ABB RAPID module: P802.mod

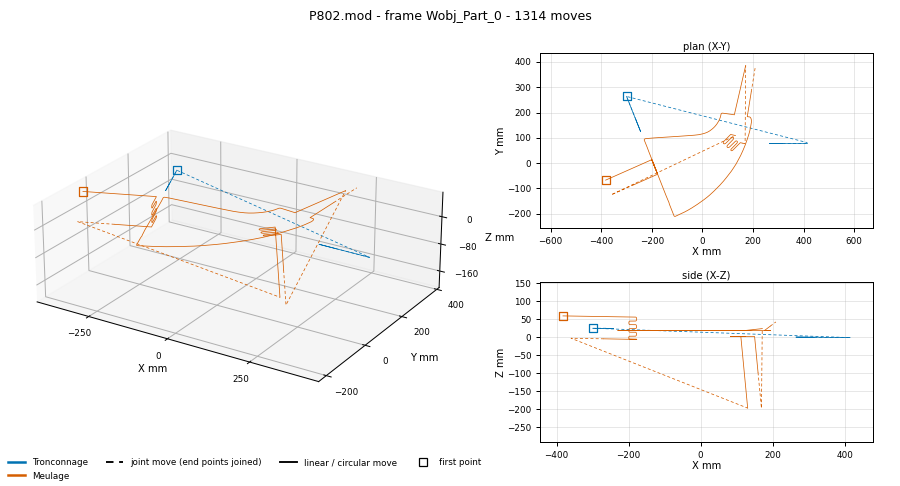
[picture p0: tool path of P802.mod in frame Wobj_Part_0, 1314 of 1328 moves have a stored position in this frame; points joined in program order, loops and branches not executed]
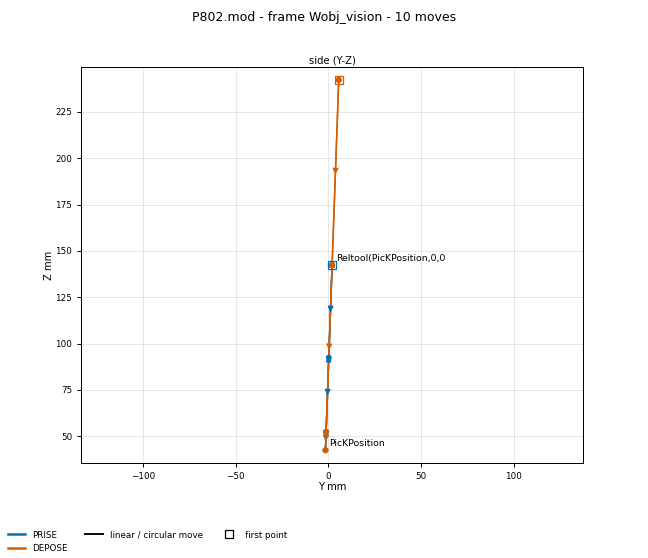
[picture p1: tool path of P802.mod in frame Wobj_vision, 10 of 1328 moves have a stored position in this frame; points joined in program order, loops and branches not executed]
MODULE P802

    ! Nom         :P802
    ! Description :
    ! Créé le     :31/05/2023 09:39:48

    LOCAL CONST SPEEDDATA VitesseLente :=[3,500,0,0];
	LOCAL CONST SPEEDDATA VitesseRapide :=[30,500,0,0];
	LOCAL CONST SPEEDDATA VitesseTronconnage :=[2,500,0,0];
	LOCAL CONST SPEEDDATA VitesseTronconnageApp :=[10,500,0,0];
    !
    !Point de prise
    LOCAL PERS Robtarget PicKPosition := [[-42.0484766120473,-1.61957801853713,42.4060496277998],[0.0147319075907155,0.941094234914177,-0.337609036243247,0.0120312325612993],[0,0,0,0],[8.999999E+09,8.999999E+09,8.999999E+09,8.999999E+09,8.999999E+09,8.999999E+09]];
	LOCAL PERS Pose Ref := [[0,0,0],[1,0,0,0]];
    !
    !Declaration des points de meulage

    !Tr_meulage_motif_1 : Meulage d'un motif
    LOCAL CONST Robtarget Tr_meulage_motif_1_0 := [[-199.5515,14.0755400390625,55.70646484375],[0.587839766788017,-0.597604018313253,0.388723125784971,-0.382371778977509],[0,0,0,0],[8.999999E+09,8.999999E+09,8.999999E+09,8.999999E+09,8.999999E+09,8.999999E+09]];
    LOCAL CONST Robtarget Tr_meulage_motif_1_1 := [[-199.1803125,13.146982421875,55.70646484375],[0.587839766788017,-0.597604018313253,0.388723125784971,-0.382371778977509],[0,0,0,0],[8.999999E+09,8.999999E+09,8.999999E+09,8.999999E+09,8.999999E+09,8.999999E+09]];
    LOCAL CONST Robtarget Tr_meulage_motif_1_2 := [[-198.809125,12.2184248046875,55.70646484375],[0.587839766788017,-0.597604018313253,0.388723125784971,-0.382371778977509],[0,0,0,0],[8.999999E+09,8.999999E+09,8.999999E+09,8.999999E+09,8.999999E+09,8.999999E+09]];
    LOCAL CONST Robtarget Tr_meulage_motif_1_3 := [[-198.4379375,11.2898671875,55.70646875],[0.587839766788017,-0.597604018313253,0.388723125784971,-0.382371778977509],[0,0,0,0],[8.999999E+09,8.999999E+09,8.999999E+09,8.999999E+09,8.999999E+09,8.999999E+09]];
    LOCAL CONST Robtarget Tr_meulage_motif_1_4 := [[-198.06675,10.36130859375,55.70646875],[0.587839766788017,-0.597604018313253,0.388723125784971,-0.382371778977509],[0,0,0,0],[8.999999E+09,8.999999E+09,8.999999E+09,8.999999E+09,8.999999E+09,8.999999E+09]];
    LOCAL CONST Robtarget Tr_meulage_motif_1_5 := [[-197.6955625,9.4327509765625,55.70646875],[0.587839766788017,-0.597604018313253,0.388723125784971,-0.382371778977509],[0,0,0,0],[8.999999E+09,8.999999E+09,8.999999E+09,8.999999E+09,8.999999E+09,8.999999E+09]];
    LOCAL CONST Robtarget Tr_meulage_motif_1_6 := [[-197.324375,8.504193359375,55.70646875],[0.587839766788017,-0.597604018313253,0.388723125784971,-0.382371778977509],[0,0,0,0],[8.999999E+09,8.999999E+09,8.999999E+09,8.999999E+09,8.999999E+09,8.999999E+09]];
    LOCAL CONST Robtarget Tr_meulage_motif_1_7 := [[-196.9531875,7.57563525390625,55.70646875],[0.587839766788017,-0.597604018313253,0.388723125784971,-0.382371778977509],[0,0,0,0],[8.999999E+09,8.999999E+09,8.999999E+09,8.999999E+09,8.999999E+09,8.999999E+09]];
    LOCAL CONST Robtarget Tr_meulage_motif_1_8 := [[-196.582,6.64707763671875,55.70647265625],[0.587839766788017,-0.597604018313253,0.388723125784971,-0.382371778977509],[0,0,0,0],[8.999999E+09,8.999999E+09,8.999999E+09,8.999999E+09,8.999999E+09,8.999999E+09]];
    LOCAL CONST Robtarget Tr_meulage_motif_1_9 := [[-196.2108125,5.71852001953125,55.70647265625],[0.587839766788017,-0.597604018313253,0.388723125784971,-0.382371778977509],[0,0,0,0],[8.999999E+09,8.999999E+09,8.999999E+09,8.999999E+09,8.999999E+09,8.999999E+09]];
    LOCAL CONST Robtarget Tr_meulage_motif_1_10 := [[-195.839625,4.7899619140625,55.70647265625],[0.587839766788017,-0.597604018313253,0.388723125784971,-0.382371778977509],[0,0,0,0],[8.999999E+09,8.999999E+09,8.999999E+09,8.999999E+09,8.999999E+09,8.999999E+09]];
    LOCAL CONST Robtarget Tr_meulage_motif_1_11 := [[-195.4684375,3.861404296875,55.70647265625],[0.587839766788017,-0.597604018313253,0.388723125784971,-0.382371778977509],[0,0,0,0],[8.999999E+09,8.999999E+09,8.999999E+09,8.999999E+09,8.999999E+09,8.999999E+09]];
    LOCAL CONST Robtarget Tr_meulage_motif_1_12 := [[-195.09725,2.93284643554688,55.70647265625],[0.587839766788017,-0.597604018313253,0.388723125784971,-0.382371778977509],[0,0,0,0],[8.999999E+09,8.999999E+09,8.999999E+09,8.999999E+09,8.999999E+09,8.999999E+09]];
    LOCAL CONST Robtarget Tr_meulage_motif_1_13 := [[-194.7260625,2.00428857421875,55.7064765625],[0.587839766788017,-0.597604018313253,0.388723125784971,-0.382371778977509],[0,0,0,0],[8.999999E+09,8.999999E+09,8.999999E+09,8.999999E+09,8.999999E+09,8.999999E+09]];
    LOCAL CONST Robtarget Tr_meulage_motif_1_14 := [[-194.354875,1.07573071289063,55.7064765625],[0.587839766788017,-0.597604018313253,0.388723125784971,-0.382371778977509],[0,0,0,0],[8.999999E+09,8.999999E+09,8.999999E+09,8.999999E+09,8.999999E+09,8.999999E+09]];
    LOCAL CONST Robtarget Tr_meulage_motif_1_15 := [[-193.9836875,0.147172897338867,55.7064765625],[0.587839766788017,-0.597604018313253,0.388723125784971,-0.382371778977509],[0,0,0,0],[8.999999E+09,8.999999E+09,8.999999E+09,8.999999E+09,8.999999E+09,8.999999E+09]];
    LOCAL CONST Robtarget Tr_meulage_motif_1_16 := [[-193.6125,-0.781384948730469,55.7064765625],[0.587839766788017,-0.597604018313253,0.388723125784971,-0.382371778977509],[0,0,0,0],[8.999999E+09,8.999999E+09,8.999999E+09,8.999999E+09,8.999999E+09,8.999999E+09]];
    LOCAL CONST Robtarget Tr_meulage_motif_1_17 := [[-193.2413125,-1.70994274902344,55.70648046875],[0.587839766788017,-0.597604018313253,0.388723125784971,-0.382371778977509],[0,0,0,0],[8.999999E+09,8.999999E+09,8.999999E+09,8.999999E+09,8.999999E+09,8.999999E+09]];
    LOCAL CONST Robtarget Tr_meulage_motif_1_18 := [[-192.870125,-2.63850048828125,55.70648046875],[0.587839766788017,-0.597604018313253,0.388723125784971,-0.382371778977509],[0,0,0,0],[8.999999E+09,8.999999E+09,8.999999E+09,8.999999E+09,8.999999E+09,8.999999E+09]];
    LOCAL CONST Robtarget Tr_meulage_motif_1_19 := [[-192.4989375,-3.56705834960938,55.70648046875],[0.587839766788017,-0.597604018313253,0.388723125784971,-0.382371778977509],[0,0,0,0],[8.999999E+09,8.999999E+09,8.999999E+09,8.999999E+09,8.999999E+09,8.999999E+09]];
    LOCAL CONST Robtarget Tr_meulage_motif_1_20 := [[-192.12775,-4.4956162109375,55.70648046875],[0.587839766788017,-0.597604018313253,0.388723125784971,-0.382371778977509],[0,0,0,0],[8.999999E+09,8.999999E+09,8.999999E+09,8.999999E+09,8.999999E+09,8.999999E+09]];
    LOCAL CONST Robtarget Tr_meulage_motif_1_21 := [[-191.7565625,-5.424173828125,55.70648046875],[0.587839766788017,-0.597604018313253,0.388723125784971,-0.382371778977509],[0,0,0,0],[8.999999E+09,8.999999E+09,8.999999E+09,8.999999E+09,8.999999E+09,8.999999E+09]];
    LOCAL CONST Robtarget Tr_meulage_motif_1_22 := [[-191.385375,-6.35273193359375,55.706484375],[0.587839766788017,-0.597604018313253,0.388723125784971,-0.382371778977509],[0,0,0,0],[8.999999E+09,8.999999E+09,8.999999E+09,8.999999E+09,8.999999E+09,8.999999E+09]];
    LOCAL CONST Robtarget Tr_meulage_motif_1_23 := [[-191.0141875,-7.28128955078125,55.706484375],[0.587839766788017,-0.597604018313253,0.388723125784971,-0.382371778977509],[0,0,0,0],[8.999999E+09,8.999999E+09,8.999999E+09,8.999999E+09,8.999999E+09,8.999999E+09]];
    LOCAL CONST Robtarget Tr_meulage_motif_1_24 := [[-190.643,-8.20984765625,55.706484375],[0.587839766788017,-0.597604018313253,0.388723125784971,-0.382371778977509],[0,0,0,0],[8.999999E+09,8.999999E+09,8.999999E+09,8.999999E+09,8.999999E+09,8.999999E+09]];
    LOCAL CONST Robtarget Tr_meulage_motif_1_25 := [[-190.2718125,-9.1384052734375,55.706484375],[0.587839766788017,-0.597604018313253,0.388723125784971,-0.382371778977509],[0,0,0,0],[8.999999E+09,8.999999E+09,8.999999E+09,8.999999E+09,8.999999E+09,8.999999E+09]];
    LOCAL CONST Robtarget Tr_meulage_motif_1_26 := [[-189.900609375,-10.066962890625,55.706484375],[0.587839766788017,-0.597604018313253,0.388723125784971,-0.382371778977509],[0,0,0,0],[8.999999E+09,8.999999E+09,8.999999E+09,8.999999E+09,8.999999E+09,8.999999E+09]];
    LOCAL CONST Robtarget Tr_meulage_motif_1_27 := [[-189.529421875,-10.9955205078125,55.70648828125],[0.587839766788017,-0.597604018313253,0.388723125784971,-0.382371778977509],[0,0,0,0],[8.999999E+09,8.999999E+09,8.999999E+09,8.999999E+09,8.999999E+09,8.999999E+09]];
    LOCAL CONST Robtarget Tr_meulage_motif_1_28 := [[-189.158234375,-11.9240791015625,55.70648828125],[0.587839766788017,-0.597604018313253,0.388723125784971,-0.382371778977509],[0,0,0,0],[8.999999E+09,8.999999E+09,8.999999E+09,8.999999E+09,8.999999E+09,8.999999E+09]];
    LOCAL CONST Robtarget Tr_meulage_motif_1_29 := [[-188.787046875,-12.85263671875,55.70648828125],[0.587839766788017,-0.597604018313253,0.388723125784971,-0.382371778977509],[0,0,0,0],[8.999999E+09,8.999999E+09,8.999999E+09,8.999999E+09,8.999999E+09,8.999999E+09]];
    LOCAL CONST Robtarget Tr_meulage_motif_1_30 := [[-188.415859375,-13.7811943359375,55.70648828125],[0.587839766788017,-0.597604018313253,0.388723125784971,-0.382371778977509],[0,0,0,0],[8.999999E+09,8.999999E+09,8.999999E+09,8.999999E+09,8.999999E+09,8.999999E+09]];
    LOCAL CONST Robtarget Tr_meulage_motif_1_31 := [[-188.044671875,-14.709751953125,55.70648828125],[0.587839766788017,-0.597604018313253,0.388723125784971,-0.382371778977509],[0,0,0,0],[8.999999E+09,8.999999E+09,8.999999E+09,8.999999E+09,8.999999E+09,8.999999E+09]];
    LOCAL CONST Robtarget Tr_meulage_motif_1_32 := [[-187.673484375,-15.638310546875,55.7064921875],[0.587839766788017,-0.597604018313253,0.388723125784971,-0.382371778977509],[0,0,0,0],[8.999999E+09,8.999999E+09,8.999999E+09,8.999999E+09,8.999999E+09,8.999999E+09]];
    LOCAL CONST Robtarget Tr_meulage_motif_1_33 := [[-187.302296875,-16.5668671875,55.7064921875],[0.587839766788017,-0.597604018313253,0.388723125784971,-0.382371778977509],[0,0,0,0],[8.999999E+09,8.999999E+09,8.999999E+09,8.999999E+09,8.999999E+09,8.999999E+09]];
    LOCAL CONST Robtarget Tr_meulage_motif_1_34 := [[-186.931109375,-17.49542578125,55.7064921875],[0.587839766788017,-0.597604018313253,0.388723125784971,-0.382371778977509],[0,0,0,0],[8.999999E+09,8.999999E+09,8.999999E+09,8.999999E+09,8.999999E+09,8.999999E+09]];
    LOCAL CONST Robtarget Tr_meulage_motif_1_35 := [[-186.559921875,-18.423984375,55.7064921875],[0.587839766788017,-0.597604018313253,0.388723125784971,-0.382371778977509],[0,0,0,0],[8.999999E+09,8.999999E+09,8.999999E+09,8.999999E+09,8.999999E+09,8.999999E+09]];
    LOCAL CONST Robtarget Tr_meulage_motif_1_36 := [[-186.188734375,-19.352541015625,55.70649609375],[0.587839766788017,-0.597604018313253,0.388723125784971,-0.382371778977509],[0,0,0,0],[8.999999E+09,8.999999E+09,8.999999E+09,8.999999E+09,8.999999E+09,8.999999E+09]];
    LOCAL CONST Robtarget Tr_meulage_motif_1_37 := [[-185.817546875,-20.281099609375,55.70649609375],[0.587839766788017,-0.597604018313253,0.388723125784971,-0.382371778977509],[0,0,0,0],[8.999999E+09,8.999999E+09,8.999999E+09,8.999999E+09,8.999999E+09,8.999999E+09]];
    LOCAL CONST Robtarget Tr_meulage_motif_1_38 := [[-185.446359375,-21.20965625,55.70649609375],[0.587839766788017,-0.597604018313253,0.388723125784971,-0.382371778977509],[0,0,0,0],[8.999999E+09,8.999999E+09,8.999999E+09,8.999999E+09,8.999999E+09,8.999999E+09]];
    LOCAL CONST Robtarget Tr_meulage_motif_1_39 := [[-185.075171875,-22.13821484375,55.70649609375],[0.587839766788017,-0.597604018313253,0.388723125784971,-0.382371778977509],[0,0,0,0],[8.999999E+09,8.999999E+09,8.999999E+09,8.999999E+09,8.999999E+09,8.999999E+09]];
    LOCAL CONST Robtarget Tr_meulage_motif_1_40 := [[-184.703984375,-23.0667734375,55.70649609375],[0.587839766788017,-0.597604018313253,0.388723125784971,-0.382371778977509],[0,0,0,0],[8.999999E+09,8.999999E+09,8.999999E+09,8.999999E+09,8.999999E+09,8.999999E+09]];
    LOCAL CONST Robtarget Tr_meulage_motif_1_41 := [[-184.332796875,-23.995330078125,55.7065],[0.587839766788017,-0.597604018313253,0.388723125784971,-0.382371778977509],[0,0,0,0],[8.999999E+09,8.999999E+09,8.999999E+09,8.999999E+09,8.999999E+09,8.999999E+09]];
    LOCAL CONST Robtarget Tr_meulage_motif_1_42 := [[-183.961609375,-24.923888671875,55.7065],[0.587839766788017,-0.597604018313253,0.388723125784971,-0.382371778977509],[0,0,0,0],[8.999999E+09,8.999999E+09,8.999999E+09,8.999999E+09,8.999999E+09,8.999999E+09]];
    LOCAL CONST Robtarget Tr_meulage_motif_1_43 := [[-183.590421875,-25.8524453125,55.7065],[0.587839766788017,-0.597604018313253,0.388723125784971,-0.382371778977509],[0,0,0,0],[8.999999E+09,8.999999E+09,8.999999E+09,8.999999E+09,8.999999E+09,8.999999E+09]];
    LOCAL CONST Robtarget Tr_meulage_motif_1_44 := [[-183.219234375,-26.78100390625,55.7065],[0.587839766788017,-0.597604018313253,0.388723125784971,-0.382371778977509],[0,0,0,0],[8.999999E+09,8.999999E+09,8.999999E+09,8.999999E+09,8.999999E+09,8.999999E+09]];
    LOCAL CONST Robtarget Tr_meulage_motif_1_45 := [[-182.848046875,-27.7095625,55.7065],[0.587839766788017,-0.597604018313253,0.388723125784971,-0.382371778977509],[0,0,0,0],[8.999999E+09,8.999999E+09,8.999999E+09,8.999999E+09,8.999999E+09,8.999999E+09]];
    LOCAL CONST Robtarget Tr_meulage_motif_1_46 := [[-182.476859375,-28.638119140625,55.70650390625],[0.587839766788017,-0.597604018313253,0.388723125784971,-0.382371778977509],[0,0,0,0],[8.999999E+09,8.999999E+09,8.999999E+09,8.999999E+09,8.999999E+09,8.999999E+09]];
    LOCAL CONST Robtarget Tr_meulage_motif_1_47 := [[-182.105671875,-29.566677734375,55.70650390625],[0.587839766788017,-0.597604018313253,0.388723125784971,-0.382371778977509],[0,0,0,0],[8.999999E+09,8.999999E+09,8.999999E+09,8.999999E+09,8.999999E+09,8.999999E+09]];
    LOCAL CONST Robtarget Tr_meulage_motif_1_48 := [[-181.734484375,-30.495234375,55.70650390625],[0.587839766788017,-0.597604018313253,0.388723125784971,-0.382371778977509],[0,0,0,0],[8.999999E+09,8.999999E+09,8.999999E+09,8.999999E+09,8.999999E+09,8.999999E+09]];
    LOCAL CONST Robtarget Tr_meulage_motif_1_49 := [[-181.363296875,-31.42379296875,55.70650390625],[0.587839766788017,-0.597604018313253,0.388723125784971,-0.382371778977509],[0,0,0,0],[8.999999E+09,8.999999E+09,8.999999E+09,8.999999E+09,8.999999E+09,8.999999E+09]];
    LOCAL CONST Robtarget Tr_meulage_motif_1_50 := [[-180.992109375,-32.3523515625,55.70650390625],[0.587839766788017,-0.597604018313253,0.388723125784971,-0.382371778977509],[0,0,0,0],[8.999999E+09,8.999999E+09,8.999999E+09,8.999999E+09,8.999999E+09,8.999999E+09]];
    LOCAL CONST Robtarget Tr_meulage_motif_1_51 := [[-180.620921875,-33.28091015625,55.7065078125],[0.587839766788017,-0.597604018313253,0.388723125784971,-0.382371778977509],[0,0,0,0],[8.999999E+09,8.999999E+09,8.999999E+09,8.999999E+09,8.999999E+09,8.999999E+09]];
    LOCAL CONST Robtarget Tr_meulage_motif_1_52 := [[-180.249734375,-34.20946484375,55.7065078125],[0.587839766788017,-0.597604018313253,0.388723125784971,-0.382371778977509],[0,0,0,0],[8.999999E+09,8.999999E+09,8.999999E+09,8.999999E+09,8.999999E+09,8.999999E+09]];
    LOCAL CONST Robtarget Tr_meulage_motif_1_53 := [[-179.8824375,-35.1315703125,55.595921875],[0.587839766788017,-0.597604018313253,0.388723125784971,-0.382371778977509],[0,0,0,0],[8.999999E+09,8.999999E+09,8.999999E+09,8.999999E+09,8.999999E+09,8.999999E+09]];
    LOCAL CONST Robtarget Tr_meulage_motif_1_54 := [[-179.53328125,-36.01131640625,55.38474609375],[0.587839766788017,-0.597604018313253,0.388723125784971,-0.382371778977509],[0,0,0,0],[8.999999E+09,8.999999E+09,8.999999E+09,8.999999E+09,8.999999E+09,8.999999E+09]];
    LOCAL CONST Robtarget Tr_meulage_motif_1_55 := [[-179.219546875,-36.80423046875,55.112921875],[0.587839766788017,-0.597604018313253,0.388723125784971,-0.382371778977509],[0,0,0,0],[8.999999E+09,8.999999E+09,8.999999E+09,8.999999E+09,8.999999E+09,8.999999E+09]];
    LOCAL CONST Robtarget Tr_meulage_motif_1_56 := [[-178.944015625,-37.50172265625,54.837],[0.587839766788017,-0.597604018313253,0.388723125784971,-0.382371778977509],[0,0,0,0],[8.999999E+09,8.999999E+09,8.999999E+09,8.999999E+09,8.999999E+09,8.999999E+09]];
    LOCAL CONST Robtarget Tr_meulage_motif_1_57 := [[-178.541625,-38.5266484375,54.2209140625],[0.587839766788017,-0.597604018313253,0.388723125784971,-0.382371778977509],[0,0,0,0],[8.999999E+09,8.999999E+09,8.999999E+09,8.999999E+09,8.999999E+09,8.999999E+09]];
    LOCAL CONST Robtarget Tr_meulage_motif_1_58 := [[-178.170265625,-39.4808515625,53.3733125],[0.587839766788017,-0.597604018313253,0.388723125784971,-0.382371778977509],[0,0,0,0],[8.999999E+09,8.999999E+09,8.999999E+09,8.999999E+09,8.999999E+09,8.999999E+09]];
    LOCAL CONST Robtarget Tr_meulage_motif_1_59 := [[-177.866125,-40.27214453125,52.3495],[0.587839766788017,-0.597604018313253,0.388723125784971,-0.382371778977509],[0,0,0,0],[8.999999E+09,8.999999E+09,8.999999E+09,8.999999E+09,8.999999E+09,8.999999E+09]];
    LOCAL CONST Robtarget Tr_meulage_motif_1_60 := [[-177.696375,-40.73000390625,51.23337890625],[0.587839766788017,-0.597604018313253,0.388723125784971,-0.382371778977509],[0,0,0,0],[8.999999E+09,8.999999E+09,8.999999E+09,8.999999E+09,8.999999E+09,8.999999E+09]];
    LOCAL CONST Robtarget Tr_meulage_motif_1_61 := [[-177.69346875,-40.757984375,50.537453125],[0.587839766788017,-0.597604018313253,0.388723125784971,-0.382371778977509],[0,0,0,0],[8.999999E+09,8.999999E+09,8.999999E+09,8.999999E+09,8.999999E+09,8.999999E+09]];
    LOCAL CONST Robtarget Tr_meulage_motif_1_62 := [[-177.70025,-40.7606953125,49.8762421875],[0.587839766788017,-0.597604018313253,0.388723125784971,-0.382371778977509],[0,0,0,0],[8.999999E+09,8.999999E+09,8.999999E+09,8.999999E+09,8.999999E+09,8.999999E+09]];
    LOCAL CONST Robtarget Tr_meulage_motif_1_63 := [[-177.727390625,-40.712453125,49.21519140625],[0.587839766788017,-0.597604018313253,0.388723125784971,-0.382371778977509],[0,0,0,0],[8.999999E+09,8.999999E+09,8.999999E+09,8.999999E+09,8.999999E+09,8.999999E+09]];
    LOCAL CONST Robtarget Tr_meulage_motif_1_64 := [[-177.923625,-40.25434375,48.1135078125],[0.587839766788017,-0.597604018313253,0.388723125784971,-0.382371778977509],[0,0,0,0],[8.999999E+09,8.999999E+09,8.999999E+09,8.999999E+09,8.999999E+09,8.999999E+09]];
    LOCAL CONST Robtarget Tr_meulage_motif_1_65 := [[-178.25190625,-39.463046875,47.10694140625],[0.587839766788017,-0.597604018313253,0.388723125784971,-0.382371778977509],[0,0,0,0],[8.999999E+09,8.999999E+09,8.999999E+09,8.999999E+09,8.999999E+09,8.999999E+09]];
    LOCAL CONST Robtarget Tr_meulage_motif_1_66 := [[-178.64028125,-38.51615234375,46.2781171875],[0.587839766788017,-0.597604018313253,0.388723125784971,-0.382371778977509],[0,0,0,0],[8.999999E+09,8.999999E+09,8.999999E+09,8.999999E+09,8.999999E+09,8.999999E+09]];
    LOCAL CONST Robtarget Tr_meulage_motif_1_67 := [[-178.899390625,-37.87976953125,45.882390625],[0.587839766788017,-0.597604018313253,0.388723125784971,-0.382371778977509],[0,0,0,0],[8.999999E+09,8.999999E+09,8.999999E+09,8.999999E+09,8.999999E+09,8.999999E+09]];
    LOCAL CONST Robtarget Tr_meulage_motif_1_68 := [[-179.33428125,-36.8063515625,45.39488671875],[0.587839766788017,-0.597604018313253,0.388723125784971,-0.382371778977509],[0,0,0,0],[8.999999E+09,8.999999E+09,8.999999E+09,8.999999E+09,8.999999E+09,8.999999E+09]];
    LOCAL CONST Robtarget Tr_meulage_motif_1_69 := [[-179.65065625,-36.0227734375,45.13080859375],[0.587839766788017,-0.597604018313253,0.388723125784971,-0.382371778977509],[0,0,0,0],[8.999999E+09,8.999999E+09,8.999999E+09,8.999999E+09,8.999999E+09,8.999999E+09]];
    LOCAL CONST Robtarget Tr_meulage_motif_1_70 := [[-179.9986875,-35.1581953125,44.9263515625],[0.587839766788017,-0.597604018313253,0.388723125784971,-0.382371778977509],[0,0,0,0],[8.999999E+09,8.999999E+09,8.999999E+09,8.999999E+09,8.999999E+09,8.999999E+09]];
    LOCAL CONST Robtarget Tr_meulage_motif_1_71 := [[-180.36415625,-34.247203125,44.817765625],[0.587839766788017,-0.597604018313253,0.388723125784971,-0.382371778977509],[0,0,0,0],[8.999999E+09,8.999999E+09,8.999999E+09,8.999999E+09,8.999999E+09,8.999999E+09]];
    LOCAL CONST Robtarget Tr_meulage_motif_1_72 := [[-180.73371875,-33.32600390625,44.70717578125],[0.587839766788017,-0.597604018313253,0.388723125784971,-0.382371778977509],[0,0,0,0],[8.999999E+09,8.999999E+09,8.999999E+09,8.999999E+09,8.999999E+09,8.999999E+09]];
    LOCAL CONST Robtarget Tr_meulage_motif_1_73 := [[-181.10490625,-32.397447265625,44.70717578125],[0.587839766788017,-0.597604018313253,0.388723125784971,-0.382371778977509],[0,0,0,0],[8.999999E+09,8.999999E+09,8.999999E+09,8.999999E+09,8.999999E+09,8.999999E+09]];
    LOCAL CONST Robtarget Tr_meulage_motif_1_74 := [[-181.47609375,-31.468890625,44.70717578125],[0.587839766788017,-0.597604018313253,0.388723125784971,-0.382371778977509],[0,0,0,0],[8.999999E+09,8.999999E+09,8.999999E+09,8.999999E+09,8.999999E+09,8.999999E+09]];
    LOCAL CONST Robtarget Tr_meulage_motif_1_75 := [[-181.84728125,-30.54033203125,44.70717578125],[0.587839766788017,-0.597604018313253,0.388723125784971,-0.382371778977509],[0,0,0,0],[8.999999E+09,8.999999E+09,8.999999E+09,8.999999E+09,8.999999E+09,8.999999E+09]];
    LOCAL CONST Robtarget Tr_meulage_motif_1_76 := [[-182.21846875,-29.6117734375,44.70717578125],[0.587839766788017,-0.597604018313253,0.388723125784971,-0.382371778977509],[0,0,0,0],[8.999999E+09,8.999999E+09,8.999999E+09,8.999999E+09,8.999999E+09,8.999999E+09]];
    LOCAL CONST Robtarget Tr_meulage_motif_1_77 := [[-182.58965625,-28.683216796875,44.707171875],[0.587839766788017,-0.597604018313253,0.388723125784971,-0.382371778977509],[0,0,0,0],[8.999999E+09,8.999999E+09,8.999999E+09,8.999999E+09,8.999999E+09,8.999999E+09]];
    LOCAL CONST Robtarget Tr_meulage_motif_1_78 := [[-182.96084375,-27.754658203125,44.707171875],[0.587839766788017,-0.597604018313253,0.388723125784971,-0.382371778977509],[0,0,0,0],[8.999999E+09,8.999999E+09,8.999999E+09,8.999999E+09,8.999999E+09,8.999999E+09]];
    LOCAL CONST Robtarget Tr_meulage_motif_1_79 := [[-183.33203125,-26.8261015625,44.707171875],[0.587839766788017,-0.597604018313253,0.388723125784971,-0.382371778977509],[0,0,0,0],[8.999999E+09,8.999999E+09,8.999999E+09,8.999999E+09,8.999999E+09,8.999999E+09]];
    LOCAL CONST Robtarget Tr_meulage_motif_1_80 := [[-183.70321875,-25.89754296875,44.707171875],[0.587839766788017,-0.597604018313253,0.388723125784971,-0.382371778977509],[0,0,0,0],[8.999999E+09,8.999999E+09,8.999999E+09,8.999999E+09,8.999999E+09,8.999999E+09]];
    LOCAL CONST Robtarget Tr_meulage_motif_1_81 := [[-184.07440625,-24.968984375,44.707171875],[0.587839766788017,-0.597604018313253,0.388723125784971,-0.382371778977509],[0,0,0,0],[8.999999E+09,8.999999E+09,8.999999E+09,8.999999E+09,8.999999E+09,8.999999E+09]];
    LOCAL CONST Robtarget Tr_meulage_motif_1_82 := [[-184.44559375,-24.040427734375,44.70716796875],[0.587839766788017,-0.597604018313253,0.388723125784971,-0.382371778977509],[0,0,0,0],[8.999999E+09,8.999999E+09,8.999999E+09,8.999999E+09,8.999999E+09,8.999999E+09]];
    LOCAL CONST Robtarget Tr_meulage_motif_1_83 := [[-184.81678125,-23.111869140625,44.70716796875],[0.587839766788017,-0.597604018313253,0.388723125784971,-0.382371778977509],[0,0,0,0],[8.999999E+09,8.999999E+09,8.999999E+09,8.999999E+09,8.999999E+09,8.999999E+09]];
    LOCAL CONST Robtarget Tr_meulage_motif_1_84 := [[-185.18796875,-22.1833125,44.70716796875],[0.587839766788017,-0.597604018313253,0.388723125784971,-0.382371778977509],[0,0,0,0],[8.999999E+09,8.999999E+09,8.999999E+09,8.999999E+09,8.999999E+09,8.999999E+09]];
    LOCAL CONST Robtarget Tr_meulage_motif_1_85 := [[-185.55915625,-21.25475390625,44.70716796875],[0.587839766788017,-0.597604018313253,0.388723125784971,-0.382371778977509],[0,0,0,0],[8.999999E+09,8.999999E+09,8.999999E+09,8.999999E+09,8.999999E+09,8.999999E+09]];
    LOCAL CONST Robtarget Tr_meulage_motif_1_86 := [[-185.93034375,-20.3261953125,44.7071640625],[0.587839766788017,-0.597604018313253,0.388723125784971,-0.382371778977509],[0,0,0,0],[8.999999E+09,8.999999E+09,8.999999E+09,8.999999E+09,8.999999E+09,8.999999E+09]];
    LOCAL CONST Robtarget Tr_meulage_motif_1_87 := [[-186.30153125,-19.397638671875,44.7071640625],[0.587839766788017,-0.597604018313253,0.388723125784971,-0.382371778977509],[0,0,0,0],[8.999999E+09,8.999999E+09,8.999999E+09,8.999999E+09,8.999999E+09,8.999999E+09]];
    LOCAL CONST Robtarget Tr_meulage_motif_1_88 := [[-186.67271875,-18.469080078125,44.7071640625],[0.587839766788017,-0.597604018313253,0.388723125784971,-0.382371778977509],[0,0,0,0],[8.999999E+09,8.999999E+09,8.999999E+09,8.999999E+09,8.999999E+09,8.999999E+09]];
    LOCAL CONST Robtarget Tr_meulage_motif_1_89 := [[-187.04390625,-17.5405234375,44.7071640625],[0.587839766788017,-0.597604018313253,0.388723125784971,-0.382371778977509],[0,0,0,0],[8.999999E+09,8.999999E+09,8.999999E+09,8.999999E+09,8.999999E+09,8.999999E+09]];
    LOCAL CONST Robtarget Tr_meulage_motif_1_90 := [[-187.41509375,-16.61196484375,44.7071640625],[0.587839766788017,-0.597604018313253,0.388723125784971,-0.382371778977509],[0,0,0,0],[8.999999E+09,8.999999E+09,8.999999E+09,8.999999E+09,8.999999E+09,8.999999E+09]];
    LOCAL CONST Robtarget Tr_meulage_motif_1_91 := [[-187.78628125,-15.6834072265625,44.70716015625],[0.587839766788017,-0.597604018313253,0.388723125784971,-0.382371778977509],[0,0,0,0],[8.999999E+09,8.999999E+09,8.999999E+09,8.999999E+09,8.999999E+09,8.999999E+09]];
    LOCAL CONST Robtarget Tr_meulage_motif_1_92 := [[-188.15746875,-14.754849609375,44.70716015625],[0.587839766788017,-0.597604018313253,0.388723125784971,-0.382371778977509],[0,0,0,0],[8.999999E+09,8.999999E+09,8.999999E+09,8.999999E+09,8.999999E+09,8.999999E+09]];
    LOCAL CONST Robtarget Tr_meulage_motif_1_93 := [[-188.52865625,-13.826291015625,44.70716015625],[0.587839766788017,-0.597604018313253,0.388723125784971,-0.382371778977509],[0,0,0,0],[8.999999E+09,8.999999E+09,8.999999E+09,8.999999E+09,8.999999E+09,8.999999E+09]];
    LOCAL CONST Robtarget Tr_meulage_motif_1_94 := [[-188.89984375,-12.8977333984375,44.70716015625],[0.587839766788017,-0.597604018313253,0.388723125784971,-0.382371778977509],[0,0,0,0],[8.999999E+09,8.999999E+09,8.999999E+09,8.999999E+09,8.999999E+09,8.999999E+09]];
    LOCAL CONST Robtarget Tr_meulage_motif_1_95 := [[-189.27103125,-11.96917578125,44.70716015625],[0.587839766788017,-0.597604018313253,0.388723125784971,-0.382371778977509],[0,0,0,0],[8.999999E+09,8.999999E+09,8.999999E+09,8.999999E+09,8.999999E+09,8.999999E+09]];
    LOCAL CONST Robtarget Tr_meulage_motif_1_96 := [[-189.64221875,-11.0406181640625,44.70715625],[0.587839766788017,-0.597604018313253,0.388723125784971,-0.382371778977509],[0,0,0,0],[8.999999E+09,8.999999E+09,8.999999E+09,8.999999E+09,8.999999E+09,8.999999E+09]];
    LOCAL CONST Robtarget Tr_meulage_motif_1_97 := [[-190.01340625,-10.1120595703125,44.70715625],[0.587839766788017,-0.597604018313253,0.388723125784971,-0.382371778977509],[0,0,0,0],[8.999999E+09,8.999999E+09,8.999999E+09,8.999999E+09,8.999999E+09,8.999999E+09]];
    LOCAL CONST Robtarget Tr_meulage_motif_1_98 := [[-190.38459375,-9.183501953125,44.70715625],[0.587839766788017,-0.597604018313253,0.388723125784971,-0.382371778977509],[0,0,0,0],[8.999999E+09,8.999999E+09,8.999999E+09,8.999999E+09,8.999999E+09,8.999999E+09]];
    LOCAL CONST Robtarget Tr_meulage_motif_1_99 := [[-190.75578125,-8.2549443359375,44.70715625],[0.587839766788017,-0.597604018313253,0.388723125784971,-0.382371778977509],[0,0,0,0],[8.999999E+09,8.999999E+09,8.999999E+09,8.999999E+09,8.999999E+09,8.999999E+09]];
    LOCAL CONST Robtarget Tr_meulage_motif_1_100 := [[-191.12696875,-7.32638671875,44.70715625],[0.587839766788017,-0.597604018313253,0.388723125784971,-0.382371778977509],[0,0,0,0],[8.999999E+09,8.999999E+09,8.999999E+09,8.999999E+09,8.999999E+09,8.999999E+09]];
    LOCAL CONST Robtarget Tr_meulage_motif_1_101 := [[-191.49815625,-6.39782861328125,44.70715234375],[0.587839766788017,-0.597604018313253,0.388723125784971,-0.382371778977509],[0,0,0,0],[8.999999E+09,8.999999E+09,8.999999E+09,8.999999E+09,8.999999E+09,8.999999E+09]];
    LOCAL CONST Robtarget Tr_meulage_motif_1_102 := [[-191.86934375,-5.46927099609375,44.70715234375],[0.587839766788017,-0.597604018313253,0.388723125784971,-0.382371778977509],[0,0,0,0],[8.999999E+09,8.999999E+09,8.999999E+09,8.999999E+09,8.999999E+09,8.999999E+09]];
    LOCAL CONST Robtarget Tr_meulage_motif_1_103 := [[-192.24053125,-4.540712890625,44.70715234375],[0.587839766788017,-0.597604018313253,0.388723125784971,-0.382371778977509],[0,0,0,0],[8.999999E+09,8.999999E+09,8.999999E+09,8.999999E+09,8.999999E+09,8.999999E+09]];
    LOCAL CONST Robtarget Tr_meulage_motif_1_104 := [[-192.61171875,-3.6121552734375,44.70715234375],[0.587839766788017,-0.597604018313253,0.388723125784971,-0.382371778977509],[0,0,0,0],[8.999999E+09,8.999999E+09,8.999999E+09,8.999999E+09,8.999999E+09,8.999999E+09]];
    LOCAL CONST Robtarget Tr_meulage_motif_1_105 := [[-192.98290625,-2.68359741210937,44.7071484375],[0.587839766788017,-0.597604018313253,0.388723125784971,-0.382371778977509],[0,0,0,0],[8.999999E+09,8.999999E+09,8.999999E+09,8.999999E+09,8.999999E+09,8.999999E+09]];
    LOCAL CONST Robtarget Tr_meulage_motif_1_106 := [[-193.35409375,-1.75503967285156,44.7071484375],[0.587839766788017,-0.597604018313253,0.388723125784971,-0.382371778977509],[0,0,0,0],[8.999999E+09,8.999999E+09,8.999999E+09,8.999999E+09,8.999999E+09,8.999999E+09]];
    LOCAL CONST Robtarget Tr_meulage_motif_1_107 := [[-193.72528125,-0.826481811523437,44.7071484375],[0.587839766788017,-0.597604018313253,0.388723125784971,-0.382371778977509],[0,0,0,0],[8.999999E+09,8.999999E+09,8.999999E+09,8.999999E+09,8.999999E+09,8.999999E+09]];
    LOCAL CONST Robtarget Tr_meulage_motif_1_108 := [[-194.09646875,0.10207600402832,44.7071484375],[0.587839766788017,-0.597604018313253,0.388723125784971,-0.382371778977509],[0,0,0,0],[8.999999E+09,8.999999E+09,8.999999E+09,8.999999E+09,8.999999E+09,8.999999E+09]];
    LOCAL CONST Robtarget Tr_meulage_motif_1_109 := [[-194.46765625,1.0306337890625,44.7071484375],[0.587839766788017,-0.597604018313253,0.388723125784971,-0.382371778977509],[0,0,0,0],[8.999999E+09,8.999999E+09,8.999999E+09,8.999999E+09,8.999999E+09,8.999999E+09]];
    LOCAL CONST Robtarget Tr_meulage_motif_1_110 := [[-194.83884375,1.95919165039063,44.70714453125],[0.587839766788017,-0.597604018313253,0.388723125784971,-0.382371778977509],[0,0,0,0],[8.999999E+09,8.999999E+09,8.999999E+09,8.999999E+09,8.999999E+09,8.999999E+09]];
    LOCAL CONST Robtarget Tr_meulage_motif_1_111 := [[-195.21003125,2.88774951171875,44.70714453125],[0.587839766788017,-0.597604018313253,0.388723125784971,-0.382371778977509],[0,0,0,0],[8.999999E+09,8.999999E+09,8.999999E+09,8.999999E+09,8.999999E+09,8.999999E+09]];
    LOCAL CONST Robtarget Tr_meulage_motif_1_112 := [[-195.58121875,3.81630737304688,44.70714453125],[0.587839766788017,-0.597604018313253,0.388723125784971,-0.382371778977509],[0,0,0,0],[8.999999E+09,8.999999E+09,8.999999E+09,8.999999E+09,8.999999E+09,8.999999E+09]];
    LOCAL CONST Robtarget Tr_meulage_motif_1_113 := [[-195.95240625,4.744865234375,44.70714453125],[0.587839766788017,-0.597604018313253,0.388723125784971,-0.382371778977509],[0,0,0,0],[8.999999E+09,8.999999E+09,8.999999E+09,8.999999E+09,8.999999E+09,8.999999E+09]];
    LOCAL CONST Robtarget Tr_meulage_motif_1_114 := [[-196.32359375,5.6734228515625,44.70714453125],[0.587839766788017,-0.597604018313253,0.388723125784971,-0.382371778977509],[0,0,0,0],[8.999999E+09,8.999999E+09,8.999999E+09,8.999999E+09,8.999999E+09,8.999999E+09]];
    LOCAL CONST Robtarget Tr_meulage_motif_1_115 := [[-196.69478125,6.60198095703125,44.707140625],[0.587839766788017,-0.597604018313253,0.388723125784971,-0.382371778977509],[0,0,0,0],[8.999999E+09,8.999999E+09,8.999999E+09,8.999999E+09,8.999999E+09,8.999999E+09]];
    LOCAL CONST Robtarget Tr_meulage_motif_1_116 := [[-197.06596875,7.53053857421875,44.707140625],[0.587839766788017,-0.597604018313253,0.388723125784971,-0.382371778977509],[0,0,0,0],[8.999999E+09,8.999999E+09,8.999999E+09,8.999999E+09,8.999999E+09,8.999999E+09]];
    LOCAL CONST Robtarget Tr_meulage_motif_1_117 := [[-197.43553125,8.4517373046875,44.5965546875],[0.587839766788017,-0.597604018313253,0.388723125784971,-0.382371778977509],[0,0,0,0],[8.999999E+09,8.999999E+09,8.999999E+09,8.999999E+09,8.999999E+09,8.999999E+09]];
    LOCAL CONST Robtarget Tr_meulage_motif_1_118 := [[-197.78903125,9.3297509765625,44.38537890625],[0.587839766788017,-0.597604018313253,0.388723125784971,-0.382371778977509],[0,0,0,0],[8.999999E+09,8.999999E+09,8.999999E+09,8.999999E+09,8.999999E+09,8.999999E+09]];
    LOCAL CONST Robtarget Tr_meulage_motif_1_119 := [[-198.10834375,10.120435546875,44.11355078125],[0.587839766788017,-0.597604018313253,0.388723125784971,-0.382371778977509],[0,0,0,0],[8.999999E+09,8.999999E+09,8.999999E+09,8.999999E+09,8.999999E+09,8.999999E+09]];
    LOCAL CONST Robtarget Tr_meulage_motif_1_120 := [[-198.3755625,10.779857421875,43.80941015625],[0.587839766788017,-0.597604018313253,0.388723125784971,-0.382371778977509],[0,0,0,0],[8.999999E+09,8.999999E+09,8.999999E+09,8.999999E+09,8.999999E+09,8.999999E+09]];
    LOCAL CONST Robtarget Tr_meulage_motif_1_121 := [[-198.766328125,11.737705078125,43.146921875],[0.587839766788017,-0.597604018313253,0.388723125784971,-0.382371778977509],[0,0,0,0],[8.999999E+09,8.999999E+09,8.999999E+09,8.999999E+09,8.999999E+09,8.999999E+09]];
    LOCAL CONST Robtarget Tr_meulage_motif_1_122 := [[-199.110359375,12.5715087890625,42.24503515625],[0.587839766788017,-0.597604018313253,0.388723125784971,-0.382371778977509],[0,0,0,0],[8.999999E+09,8.999999E+09,8.999999E+09,8.999999E+09,8.999999E+09,8.999999E+09]];
    LOCAL CONST Robtarget Tr_meulage_motif_1_123 := [[-199.319671875,13.0639697265625,41.1990703125],[0.587839766788017,-0.597604018313253,0.388723125784971,-0.382371778977509],[0,0,0,0],[8.999999E+09,8.999999E+09,8.999999E+09,8.999999E+09,8.999999E+09,8.999999E+09]];
    LOCAL CONST Robtarget Tr_meulage_motif_1_124 := [[-199.395359375,13.23270703125,40.505890625],[0.587839766788017,-0.597604018313253,0.388723125784971,-0.382371778977509],[0,0,0,0],[8.999999E+09,8.999999E+09,8.999999E+09,8.999999E+09,8.999999E+09,8.999999E+09]];
    LOCAL CONST Robtarget Tr_meulage_motif_1_125 := [[-199.426953125,13.2888330078125,39.7359375],[0.587839766788017,-0.597604018313253,0.388723125784971,-0.382371778977509],[0,0,0,0],[8.999999E+09,8.999999E+09,8.999999E+09,8.999999E+09,8.999999E+09,8.999999E+09]];
    LOCAL CONST Robtarget Tr_meulage_motif_1_126 := [[-199.41,13.223521484375,38.966109375],[0.587839766788017,-0.597604018313253,0.388723125784971,-0.382371778977509],[0,0,0,0],[8.999999E+09,8.999999E+09,8.999999E+09,8.999999E+09,8.999999E+09,8.999999E+09]];
    LOCAL CONST Robtarget Tr_meulage_motif_1_127 := [[-199.265625,12.829361328125,37.8579296875],[0.587839766788017,-0.597604018313253,0.388723125784971,-0.382371778977509],[0,0,0,0],[8.999999E+09,8.999999E+09,8.999999E+09,8.999999E+09,8.999999E+09,8.999999E+09]];
    LOCAL CONST Robtarget Tr_meulage_motif_1_128 := [[-199.11784375,12.4422470703125,37.27227734375],[0.587839766788017,-0.597604018313253,0.388723125784971,-0.382371778977509],[0,0,0,0],[8.999999E+09,8.999999E+09,8.999999E+09,8.999999E+09,8.999999E+09,8.999999E+09]];
    LOCAL CONST Robtarget Tr_meulage_motif_1_129 := [[-198.797640625,11.61486328125,36.38520703125],[0.587839766788017,-0.597604018313253,0.388723125784971,-0.382371778977509],[0,0,0,0],[8.999999E+09,8.999999E+09,8.999999E+09,8.999999E+09,8.999999E+09,8.999999E+09]];
    LOCAL CONST Robtarget Tr_meulage_motif_1_130 := [[-198.584484375,11.0693193359375,35.970921875],[0.587839766788017,-0.597604018313253,0.388723125784971,-0.382371778977509],[0,0,0,0],[8.999999E+09,8.999999E+09,8.999999E+09,8.999999E+09,8.999999E+09,8.999999E+09]];
    LOCAL CONST Robtarget Tr_meulage_motif_1_131 := [[-198.175109375,10.029048828125,35.426859375],[0.587839766788017,-0.597604018313253,0.388723125784971,-0.382371778977509],[0,0,0,0],[8.999999E+09,8.999999E+09,8.999999E+09,8.999999E+09,8.999999E+09,8.999999E+09]];
    LOCAL CONST Robtarget Tr_meulage_motif_1_132 := [[-197.871703125,9.2612255859375,35.13137890625],[0.587839766788017,-0.597604018313253,0.388723125784971,-0.382371778977509],[0,0,0,0],[8.999999E+09,8.999999E+09,8.999999E+09,8.999999E+09,8.999999E+09,8.999999E+09]];
    LOCAL CONST Robtarget Tr_meulage_motif_1_133 := [[-197.52784375,8.3949716796875,34.92692578125],[0.587839766788017,-0.597604018313253,0.388723125784971,-0.382371778977509],[0,0,0,0],[8.999999E+09,8.999999E+09,8.999999E+09,8.999999E+09,8.999999E+09,8.999999E+09]];
    LOCAL CONST Robtarget Tr_meulage_motif_1_134 := [[-197.164609375,7.4830888671875,34.81833984375],[0.587839766788017,-0.597604018313253,0.388723125784971,-0.382371778977509],[0,0,0,0],[8.999999E+09,8.999999E+09,8.999999E+09,8.999999E+09,8.999999E+09,8.999999E+09]];
    LOCAL CONST Robtarget Tr_meulage_motif_1_135 := [[-196.797328125,6.5609833984375,34.70775],[0.587839766788017,-0.597604018313253,0.388723125784971,-0.382371778977509],[0,0,0,0],[8.999999E+09,8.999999E+09,8.999999E+09,8.999999E+09,8.999999E+09,8.999999E+09]];
    LOCAL CONST Robtarget Tr_meulage_motif_1_136 := [[-196.426140625,5.63242578125,34.70775390625],[0.587839766788017,-0.597604018313253,0.388723125784971,-0.382371778977509],[0,0,0,0],[8.999999E+09,8.999999E+09,8.999999E+09,8.999999E+09,8.999999E+09,8.999999E+09]];
    LOCAL CONST Robtarget Tr_meulage_motif_1_137 := [[-196.054953125,4.7038681640625,34.70775390625],[0.587839766788017,-0.597604018313253,0.388723125784971,-0.382371778977509],[0,0,0,0],[8.999999E+09,8.999999E+09,8.999999E+09,8.999999E+09,8.999999E+09,8.999999E+09]];
    LOCAL CONST Robtarget Tr_meulage_motif_1_138 := [[-195.683765625,3.77531005859375,34.70775390625],[0.587839766788017,-0.597604018313253,0.388723125784971,-0.382371778977509],[0,0,0,0],[8.999999E+09,8.999999E+09,8.999999E+09,8.999999E+09,8.999999E+09,8.999999E+09]];
    LOCAL CONST Robtarget Tr_meulage_motif_1_139 := [[-195.312578125,2.84675219726563,34.70775390625],[0.587839766788017,-0.597604018313253,0.388723125784971,-0.382371778977509],[0,0,0,0],[8.999999E+09,8.999999E+09,8.999999E+09,8.999999E+09,8.999999E+09,8.999999E+09]];
    LOCAL CONST Robtarget Tr_meulage_motif_1_140 := [[-194.941390625,1.91819445800781,34.70775390625],[0.587839766788017,-0.597604018313253,0.388723125784971,-0.382371778977509],[0,0,0,0],[8.999999E+09,8.999999E+09,8.999999E+09,8.999999E+09,8.999999E+09,8.999999E+09]];
    LOCAL CONST Robtarget Tr_meulage_motif_1_141 := [[-194.570203125,0.989636657714844,34.7077578125],[0.587839766788017,-0.597604018313253,0.388723125784971,-0.382371778977509],[0,0,0,0],[8.999999E+09,8.999999E+09,8.999999E+09,8.999999E+09,8.999999E+09,8.999999E+09]];
    LOCAL CONST Robtarget Tr_meulage_motif_1_142 := [[-194.199,0.0610788383483887,34.7077578125],[0.587839766788017,-0.597604018313253,0.388723125784971,-0.382371778977509],[0,0,0,0],[8.999999E+09,8.999999E+09,8.999999E+09,8.999999E+09,8.999999E+09,8.999999E+09]];
    LOCAL CONST Robtarget Tr_meulage_motif_1_143 := [[-193.8278125,-0.86747900390625,34.7077578125],[0.587839766788017,-0.597604018313253,0.388723125784971,-0.382371778977509],[0,0,0,0],[8.999999E+09,8.999999E+09,8.999999E+09,8.999999E+09,8.999999E+09,8.999999E+09]];
    LOCAL CONST Robtarget Tr_meulage_motif_1_144 := [[-193.456625,-1.79603674316406,34.7077578125],[0.587839766788017,-0.597604018313253,0.388723125784971,-0.382371778977509],[0,0,0,0],[8.999999E+09,8.999999E+09,8.999999E+09,8.999999E+09,8.999999E+09,8.999999E+09]];
    LOCAL CONST Robtarget Tr_meulage_motif_1_145 := [[-193.0854375,-2.7245947265625,34.70776171875],[0.587839766788017,-0.597604018313253,0.388723125784971,-0.382371778977509],[0,0,0,0],[8.999999E+09,8.999999E+09,8.999999E+09,8.999999E+09,8.999999E+09,8.999999E+09]];
    LOCAL CONST Robtarget Tr_meulage_motif_1_146 := [[-192.71425,-3.65315234375,34.70776171875],[0.587839766788017,-0.597604018313253,0.388723125784971,-0.382371778977509],[0,0,0,0],[8.999999E+09,8.999999E+09,8.999999E+09,8.999999E+09,8.999999E+09,8.999999E+09]];
    LOCAL CONST Robtarget Tr_meulage_motif_1_147 := [[-192.3430625,-4.58171044921875,34.70776171875],[0.587839766788017,-0.597604018313253,0.388723125784971,-0.382371778977509],[0,0,0,0],[8.999999E+09,8.999999E+09,8.999999E+09,8.999999E+09,8.999999E+09,8.999999E+09]];
    LOCAL CONST Robtarget Tr_meulage_motif_1_148 := [[-191.971875,-5.51026806640625,34.70776171875],[0.587839766788017,-0.597604018313253,0.388723125784971,-0.382371778977509],[0,0,0,0],[8.999999E+09,8.999999E+09,8.999999E+09,8.999999E+09,8.999999E+09,8.999999E+09]];
    LOCAL CONST Robtarget Tr_meulage_motif_1_149 := [[-191.6006875,-6.43882568359375,34.70776171875],[0.587839766788017,-0.597604018313253,0.388723125784971,-0.382371778977509],[0,0,0,0],[8.999999E+09,8.999999E+09,8.999999E+09,8.999999E+09,8.999999E+09,8.999999E+09]];
    LOCAL CONST Robtarget Tr_meulage_motif_1_150 := [[-191.2295,-7.3673837890625,34.707765625],[0.587839766788017,-0.597604018313253,0.388723125784971,-0.382371778977509],[0,0,0,0],[8.999999E+09,8.999999E+09,8.999999E+09,8.999999E+09,8.999999E+09,8.999999E+09]];
    LOCAL CONST Robtarget Tr_meulage_motif_1_151 := [[-190.8583125,-8.29594140625,34.707765625],[0.587839766788017,-0.597604018313253,0.388723125784971,-0.382371778977509],[0,0,0,0],[8.999999E+09,8.999999E+09,8.999999E+09,8.999999E+09,8.999999E+09,8.999999E+09]];
    LOCAL CONST Robtarget Tr_meulage_motif_1_152 := [[-190.487125,-9.2244990234375,34.707765625],[0.587839766788017,-0.597604018313253,0.388723125784971,-0.382371778977509],[0,0,0,0],[8.999999E+09,8.999999E+09,8.999999E+09,8.999999E+09,8.999999E+09,8.999999E+09]];
    LOCAL CONST Robtarget Tr_meulage_motif_1_153 := [[-190.1159375,-10.1530576171875,34.707765625],[0.587839766788017,-0.597604018313253,0.388723125784971,-0.382371778977509],[0,0,0,0],[8.999999E+09,8.999999E+09,8.999999E+09,8.999999E+09,8.999999E+09,8.999999E+09]];
    LOCAL CONST Robtarget Tr_meulage_motif_1_154 := [[-189.74475,-11.081615234375,34.707765625],[0.587839766788017,-0.597604018313253,0.388723125784971,-0.382371778977509],[0,0,0,0],[8.999999E+09,8.999999E+09,8.999999E+09,8.999999E+09,8.999999E+09,8.999999E+09]];
    LOCAL CONST Robtarget Tr_meulage_motif_1_155 := [[-189.3735625,-12.0101728515625,34.70776953125],[0.587839766788017,-0.597604018313253,0.388723125784971,-0.382371778977509],[0,0,0,0],[8.999999E+09,8.999999E+09,8.999999E+09,8.999999E+09,8.999999E+09,8.999999E+09]];
    LOCAL CONST Robtarget Tr_meulage_motif_1_156 := [[-189.002375,-12.93873046875,34.70776953125],[0.587839766788017,-0.597604018313253,0.388723125784971,-0.382371778977509],[0,0,0,0],[8.999999E+09,8.999999E+09,8.999999E+09,8.999999E+09,8.999999E+09,8.999999E+09]];
    LOCAL CONST Robtarget Tr_meulage_motif_1_157 := [[-188.6311875,-13.8672880859375,34.70776953125],[0.587839766788017,-0.597604018313253,0.388723125784971,-0.382371778977509],[0,0,0,0],[8.999999E+09,8.999999E+09,8.999999E+09,8.999999E+09,8.999999E+09,8.999999E+09]];
    LOCAL CONST Robtarget Tr_meulage_motif_1_158 := [[-188.26,-14.7958466796875,34.70776953125],[0.587839766788017,-0.597604018313253,0.388723125784971,-0.382371778977509],[0,0,0,0],[8.999999E+09,8.999999E+09,8.999999E+09,8.999999E+09,8.999999E+09,8.999999E+09]];
    LOCAL CONST Robtarget Tr_meulage_motif_1_159 := [[-187.8888125,-15.724404296875,34.70776953125],[0.587839766788017,-0.597604018313253,0.388723125784971,-0.382371778977509],[0,0,0,0],[8.999999E+09,8.999999E+09,8.999999E+09,8.999999E+09,8.999999E+09,8.999999E+09]];
    LOCAL CONST Robtarget Tr_meulage_motif_1_160 := [[-187.517625,-16.652962890625,34.7077734375],[0.587839766788017,-0.597604018313253,0.388723125784971,-0.382371778977509],[0,0,0,0],[8.999999E+09,8.999999E+09,8.999999E+09,8.999999E+09,8.999999E+09,8.999999E+09]];
    LOCAL CONST Robtarget Tr_meulage_motif_1_161 := [[-187.1464375,-17.58151953125,34.7077734375],[0.587839766788017,-0.597604018313253,0.388723125784971,-0.382371778977509],[0,0,0,0],[8.999999E+09,8.999999E+09,8.999999E+09,8.999999E+09,8.999999E+09,8.999999E+09]];
    LOCAL CONST Robtarget Tr_meulage_motif_1_162 := [[-186.77525,-18.510078125,34.7077734375],[0.587839766788017,-0.597604018313253,0.388723125784971,-0.382371778977509],[0,0,0,0],[8.999999E+09,8.999999E+09,8.999999E+09,8.999999E+09,8.999999E+09,8.999999E+09]];
    LOCAL CONST Robtarget Tr_meulage_motif_1_163 := [[-186.4040625,-19.438634765625,34.7077734375],[0.587839766788017,-0.597604018313253,0.388723125784971,-0.382371778977509],[0,0,0,0],[8.999999E+09,8.999999E+09,8.999999E+09,8.999999E+09,8.999999E+09,8.999999E+09]];
    LOCAL CONST Robtarget Tr_meulage_motif_1_164 := [[-186.032875,-20.367193359375,34.70777734375],[0.587839766788017,-0.597604018313253,0.388723125784971,-0.382371778977509],[0,0,0,0],[8.999999E+09,8.999999E+09,8.999999E+09,8.999999E+09,8.999999E+09,8.999999E+09]];
    LOCAL CONST Robtarget Tr_meulage_motif_1_165 := [[-185.6616875,-21.295751953125,34.70777734375],[0.587839766788017,-0.597604018313253,0.388723125784971,-0.382371778977509],[0,0,0,0],[8.999999E+09,8.999999E+09,8.999999E+09,8.999999E+09,8.999999E+09,8.999999E+09]];
    LOCAL CONST Robtarget Tr_meulage_motif_1_166 := [[-185.2905,-22.22430859375,34.70777734375],[0.587839766788017,-0.597604018313253,0.388723125784971,-0.382371778977509],[0,0,0,0],[8.999999E+09,8.999999E+09,8.999999E+09,8.999999E+09,8.999999E+09,8.999999E+09]];
    LOCAL CONST Robtarget Tr_meulage_motif_1_167 := [[-184.9193125,-23.1528671875,34.70777734375],[0.587839766788017,-0.597604018313253,0.388723125784971,-0.382371778977509],[0,0,0,0],[8.999999E+09,8.999999E+09,8.999999E+09,8.999999E+09,8.999999E+09,8.999999E+09]];
    LOCAL CONST Robtarget Tr_meulage_motif_1_168 := [[-184.548125,-24.081423828125,34.70777734375],[0.587839766788017,-0.597604018313253,0.388723125784971,-0.382371778977509],[0,0,0,0],[8.999999E+09,8.999999E+09,8.999999E+09,8.999999E+09,8.999999E+09,8.999999E+09]];
    LOCAL CONST Robtarget Tr_meulage_motif_1_169 := [[-184.1769375,-25.009982421875,34.70778125],[0.587839766788017,-0.597604018313253,0.388723125784971,-0.382371778977509],[0,0,0,0],[8.999999E+09,8.999999E+09,8.999999E+09,8.999999E+09,8.999999E+09,8.999999E+09]];
    LOCAL CONST Robtarget Tr_meulage_motif_1_170 := [[-183.80575,-25.938541015625,34.70778125],[0.587839766788017,-0.597604018313253,0.388723125784971,-0.382371778977509],[0,0,0,0],[8.999999E+09,8.999999E+09,8.999999E+09,8.999999E+09,8.999999E+09,8.999999E+09]];
    LOCAL CONST Robtarget Tr_meulage_motif_1_171 := [[-183.4345625,-26.86709765625,34.70778125],[0.587839766788017,-0.597604018313253,0.388723125784971,-0.382371778977509],[0,0,0,0],[8.999999E+09,8.999999E+09,8.999999E+09,8.999999E+09,8.999999E+09,8.999999E+09]];
    LOCAL CONST Robtarget Tr_meulage_motif_1_172 := [[-183.063375,-27.79565625,34.70778125],[0.587839766788017,-0.597604018313253,0.388723125784971,-0.382371778977509],[0,0,0,0],[8.999999E+09,8.999999E+09,8.999999E+09,8.999999E+09,8.999999E+09,8.999999E+09]];
    LOCAL CONST Robtarget Tr_meulage_motif_1_173 := [[-182.6921875,-28.724212890625,34.70778125],[0.587839766788017,-0.597604018313253,0.388723125784971,-0.382371778977509],[0,0,0,0],[8.999999E+09,8.999999E+09,8.999999E+09,8.999999E+09,8.999999E+09,8.999999E+09]];
    LOCAL CONST Robtarget Tr_meulage_motif_1_174 := [[-182.321,-29.652771484375,34.70778515625],[0.587839766788017,-0.597604018313253,0.388723125784971,-0.382371778977509],[0,0,0,0],[8.999999E+09,8.999999E+09,8.999999E+09,8.999999E+09,8.999999E+09,8.999999E+09]];
    LOCAL CONST Robtarget Tr_meulage_motif_1_175 := [[-181.9498125,-30.581330078125,34.70778515625],[0.587839766788017,-0.597604018313253,0.388723125784971,-0.382371778977509],[0,0,0,0],[8.999999E+09,8.999999E+09,8.999999E+09,8.999999E+09,8.999999E+09,8.999999E+09]];
    LOCAL CONST Robtarget Tr_meulage_motif_1_176 := [[-181.578625,-31.50988671875,34.70778515625],[0.587839766788017,-0.597604018313253,0.388723125784971,-0.382371778977509],[0,0,0,0],[8.999999E+09,8.999999E+09,8.999999E+09,8.999999E+09,8.999999E+09,8.999999E+09]];
    LOCAL CONST Robtarget Tr_meulage_motif_1_177 := [[-181.2074375,-32.4384453125,34.70778515625],[0.587839766788017,-0.597604018313253,0.388723125784971,-0.382371778977509],[0,0,0,0],[8.999999E+09,8.999999E+09,8.999999E+09,8.999999E+09,8.999999E+09,8.999999E+09]];
    LOCAL CONST Robtarget Tr_meulage_motif_1_178 := [[-180.83625,-33.36700390625,34.70778515625],[0.587839766788017,-0.597604018313253,0.388723125784971,-0.382371778977509],[0,0,0,0],[8.999999E+09,8.999999E+09,8.999999E+09,8.999999E+09,8.999999E+09,8.999999E+09]];
    LOCAL CONST Robtarget Tr_meulage_motif_1_179 := [[-180.4650625,-34.2955625,34.7077890625],[0.587839766788017,-0.597604018313253,0.388723125784971,-0.382371778977509],[0,0,0,0],[8.999999E+09,8.999999E+09,8.999999E+09,8.999999E+09,8.999999E+09,8.999999E+09]];
    LOCAL CONST Robtarget Tr_meulage_motif_1_180 := [[-180.097765625,-35.2176640625,34.597203125],[0.587839766788017,-0.597604018313253,0.388723125784971,-0.382371778977509],[0,0,0,0],[8.999999E+09,8.999999E+09,8.999999E+09,8.999999E+09,8.999999E+09,8.999999E+09]];
    LOCAL CONST Robtarget Tr_meulage_motif_1_181 := [[-179.748609375,-36.09741015625,34.38602734375],[0.587839766788017,-0.597604018313253,0.388723125784971,-0.382371778977509],[0,0,0,0],[8.999999E+09,8.999999E+09,8.999999E+09,8.999999E+09,8.999999E+09,8.999999E+09]];
    LOCAL CONST Robtarget Tr_meulage_motif_1_182 := [[-179.434875,-36.89032421875,34.114203125],[0.587839766788017,-0.597604018313253,0.388723125784971,-0.382371778977509],[0,0,0,0],[8.999999E+09,8.999999E+09,8.999999E+09,8.999999E+09,8.999999E+09,8.999999E+09]];
    LOCAL CONST Robtarget Tr_meulage_motif_1_183 := [[-179.159328125,-37.58781640625,33.83828125],[0.587839766788017,-0.597604018313253,0.388723125784971,-0.382371778977509],[0,0,0,0],[8.999999E+09,8.999999E+09,8.999999E+09,8.999999E+09,8.999999E+09,8.999999E+09]];
    LOCAL CONST Robtarget Tr_meulage_motif_1_184 := [[-178.756953125,-38.6127421875,33.2221953125],[0.587839766788017,-0.597604018313253,0.388723125784971,-0.382371778977509],[0,0,0,0],[8.999999E+09,8.999999E+09,8.999999E+09,8.999999E+09,8.999999E+09,8.999999E+09]];
    LOCAL CONST Robtarget Tr_meulage_motif_1_185 := [[-178.38559375,-39.5669453125,32.374591796875],[0.587839766788017,-0.597604018313253,0.388723125784971,-0.382371778977509],[0,0,0,0],[8.999999E+09,8.999999E+09,8.999999E+09,8.999999E+09,8.999999E+09,8.999999E+09]];
    LOCAL CONST Robtarget Tr_meulage_motif_1_186 := [[-178.081453125,-40.35823828125,31.350779296875],[0.587839766788017,-0.597604018313253,0.388723125784971,-0.382371778977509],[0,0,0,0],[8.999999E+09,8.999999E+09,8.999999E+09,8.999999E+09,8.999999E+09,8.999999E+09]];
    LOCAL CONST Robtarget Tr_meulage_motif_1_187 := [[-177.911703125,-40.81609765625,30.23466015625],[0.587839766788017,-0.597604018313253,0.388723125784971,-0.382371778977509],[0,0,0,0],[8.999999E+09,8.999999E+09,8.999999E+09,8.999999E+09,8.999999E+09,8.999999E+09]];
    LOCAL CONST Robtarget Tr_meulage_motif_1_188 := [[-177.90878125,-40.844078125,29.538734375],[0.587839766788017,-0.597604018313253,0.388723125784971,-0.382371778977509],[0,0,0,0],[8.999999E+09,8.999999E+09,8.999999E+09,8.999999E+09,8.999999E+09,8.999999E+09]];
    LOCAL CONST Robtarget Tr_meulage_motif_1_189 := [[-177.9155625,-40.8467890625,28.8775234375],[0.587839766788017,-0.597604018313253,0.388723125784971,-0.382371778977509],[0,0,0,0],[8.999999E+09,8.999999E+09,8.999999E+09,8.999999E+09,8.999999E+09,8.999999E+09]];
    LOCAL CONST Robtarget Tr_meulage_motif_1_190 := [[-177.94271875,-40.798546875,28.216470703125],[0.587839766788017,-0.597604018313253,0.388723125784971,-0.382371778977509],[0,0,0,0],[8.999999E+09,8.999999E+09,8.999999E+09,8.999999E+09,8.999999E+09,8.999999E+09]];
    LOCAL CONST Robtarget Tr_meulage_motif_1_191 := [[-178.138953125,-40.3404375,27.114787109375],[0.587839766788017,-0.597604018313253,0.388723125784971,-0.382371778977509],[0,0,0,0],[8.999999E+09,8.999999E+09,8.999999E+09,8.999999E+09,8.999999E+09,8.999999E+09]];
    LOCAL CONST Robtarget Tr_meulage_motif_1_192 := [[-178.467234375,-39.549140625,26.10822265625],[0.587839766788017,-0.597604018313253,0.388723125784971,-0.382371778977509],[0,0,0,0],[8.999999E+09,8.999999E+09,8.999999E+09,8.999999E+09,8.999999E+09,8.999999E+09]];
    LOCAL CONST Robtarget Tr_meulage_motif_1_193 := [[-178.855609375,-38.60224609375,25.2793984375],[0.587839766788017,-0.597604018313253,0.388723125784971,-0.382371778977509],[0,0,0,0],[8.999999E+09,8.999999E+09,8.999999E+09,8.999999E+09,8.999999E+09,8.999999E+09]];
    LOCAL CONST Robtarget Tr_meulage_motif_1_194 := [[-179.114703125,-37.96586328125,24.883671875],[0.587839766788017,-0.597604018313253,0.388723125784971,-0.382371778977509],[0,0,0,0],[8.999999E+09,8.999999E+09,8.999999E+09,8.999999E+09,8.999999E+09,8.999999E+09]];
    LOCAL CONST Robtarget Tr_meulage_motif_1_195 := [[-179.54959375,-36.8924453125,24.396169921875],[0.587839766788017,-0.597604018313253,0.388723125784971,-0.382371778977509],[0,0,0,0],[8.999999E+09,8.999999E+09,8.999999E+09,8.999999E+09,8.999999E+09,8.999999E+09]];
    LOCAL CONST Robtarget Tr_meulage_motif_1_196 := [[-179.86596875,-36.1088671875,24.13208984375],[0.587839766788017,-0.597604018313253,0.388723125784971,-0.382371778977509],[0,0,0,0],[8.999999E+09,8.999999E+09,8.999999E+09,8.999999E+09,8.999999E+09,8.999999E+09]];
    LOCAL CONST Robtarget Tr_meulage_motif_1_197 := [[-180.214015625,-35.2442890625,23.9276328125],[0.587839766788017,-0.597604018313253,0.388723125784971,-0.382371778977509],[0,0,0,0],[8.999999E+09,8.999999E+09,8.999999E+09,8.999999E+09,8.999999E+09,8.999999E+09]];
    LOCAL CONST Robtarget Tr_meulage_motif_1_198 := [[-180.57946875,-34.333296875,23.819044921875],[0.587839766788017,-0.597604018313253,0.388723125784971,-0.382371778977509],[0,0,0,0],[8.999999E+09,8.999999E+09,8.999999E+09,8.999999E+09,8.999999E+09,8.999999E+09]];
    LOCAL CONST Robtarget Tr_meulage_motif_1_199 := [[-180.94903125,-33.4121015625,23.70845703125],[0.587839766788017,-0.597604018313253,0.388723125784971,-0.382371778977509],[0,0,0,0],[8.999999E+09,8.999999E+09,8.999999E+09,8.999999E+09,8.999999E+09,8.999999E+09]];
    LOCAL CONST Robtarget Tr_meulage_motif_1_200 := [[-181.32021875,-32.483541015625,23.70845703125],[0.587839766788017,-0.597604018313253,0.388723125784971,-0.382371778977509],[0,0,0,0],[8.999999E+09,8.999999E+09,8.999999E+09,8.999999E+09,8.999999E+09,8.999999E+09]];
    LOCAL CONST Robtarget Tr_meulage_motif_1_201 := [[-181.69140625,-31.554984375,23.70845703125],[0.587839766788017,-0.597604018313253,0.388723125784971,-0.382371778977509],[0,0,0,0],[8.999999E+09,8.999999E+09,8.999999E+09,8.999999E+09,8.999999E+09,8.999999E+09]];
    LOCAL CONST Robtarget Tr_meulage_motif_1_202 := [[-182.06259375,-30.62642578125,23.708455078125],[0.587839766788017,-0.597604018313253,0.388723125784971,-0.382371778977509],[0,0,0,0],[8.999999E+09,8.999999E+09,8.999999E+09,8.999999E+09,8.999999E+09,8.999999E+09]];
    LOCAL CONST Robtarget Tr_meulage_motif_1_203 := [[-182.43378125,-29.697869140625,23.708455078125],[0.587839766788017,-0.597604018313253,0.388723125784971,-0.382371778977509],[0,0,0,0],[8.999999E+09,8.999999E+09,8.999999E+09,8.999999E+09,8.999999E+09,8.999999E+09]];
    LOCAL CONST Robtarget Tr_meulage_motif_1_204 := [[-182.80496875,-28.769310546875,23.708453125],[0.587839766788017,-0.597604018313253,0.388723125784971,-0.382371778977509],[0,0,0,0],[8.999999E+09,8.999999E+09,8.999999E+09,8.999999E+09,8.999999E+09,8.999999E+09]];
    LOCAL CONST Robtarget Tr_meulage_motif_1_205 := [[-183.17615625,-27.840751953125,23.708453125],[0.587839766788017,-0.597604018313253,0.388723125784971,-0.382371778977509],[0,0,0,0],[8.999999E+09,8.999999E+09,8.999999E+09,8.999999E+09,8.999999E+09,8.999999E+09]];
    LOCAL CONST Robtarget Tr_meulage_motif_1_206 := [[-183.54734375,-26.9121953125,23.708451171875],[0.587839766788017,-0.597604018313253,0.388723125784971,-0.382371778977509],[0,0,0,0],[8.999999E+09,8.999999E+09,8.999999E+09,8.999999E+09,8.999999E+09,8.999999E+09]];
    LOCAL CONST Robtarget Tr_meulage_motif_1_207 := [[-183.918546875,-25.98363671875,23.708451171875],[0.587839766788017,-0.597604018313253,0.388723125784971,-0.382371778977509],[0,0,0,0],[8.999999E+09,8.999999E+09,8.999999E+09,8.999999E+09,8.999999E+09,8.999999E+09]];
    LOCAL CONST Robtarget Tr_meulage_motif_1_208 := [[-184.289734375,-25.055080078125,23.708451171875],[0.587839766788017,-0.597604018313253,0.388723125784971,-0.382371778977509],[0,0,0,0],[8.999999E+09,8.999999E+09,8.999999E+09,8.999999E+09,8.999999E+09,8.999999E+09]];
    LOCAL CONST Robtarget Tr_meulage_motif_1_209 := [[-184.660921875,-24.126521484375,23.70844921875],[0.587839766788017,-0.597604018313253,0.388723125784971,-0.382371778977509],[0,0,0,0],[8.999999E+09,8.999999E+09,8.999999E+09,8.999999E+09,8.999999E+09,8.999999E+09]];
    LOCAL CONST Robtarget Tr_meulage_motif_1_210 := [[-185.032109375,-23.197962890625,23.70844921875],[0.587839766788017,-0.597604018313253,0.388723125784971,-0.382371778977509],[0,0,0,0],[8.999999E+09,8.999999E+09,8.999999E+09,8.999999E+09,8.999999E+09,8.999999E+09]];
    LOCAL CONST Robtarget Tr_meulage_motif_1_211 := [[-185.403296875,-22.26940625,23.708447265625],[0.587839766788017,-0.597604018313253,0.388723125784971,-0.382371778977509],[0,0,0,0],[8.999999E+09,8.999999E+09,8.999999E+09,8.999999E+09,8.999999E+09,8.999999E+09]];
    LOCAL CONST Robtarget Tr_meulage_motif_1_212 := [[-185.774484375,-21.34084765625,23.708447265625],[0.587839766788017,-0.597604018313253,0.388723125784971,-0.382371778977509],[0,0,0,0],[8.999999E+09,8.999999E+09,8.999999E+09,8.999999E+09,8.999999E+09,8.999999E+09]];
    LOCAL CONST Robtarget Tr_meulage_motif_1_213 := [[-186.145671875,-20.412291015625,23.708447265625],[0.587839766788017,-0.597604018313253,0.388723125784971,-0.382371778977509],[0,0,0,0],[8.999999E+09,8.999999E+09,8.999999E+09,8.999999E+09,8.999999E+09,8.999999E+09]];
    LOCAL CONST Robtarget Tr_meulage_motif_1_214 := [[-186.516859375,-19.483732421875,23.7084453125],[0.587839766788017,-0.597604018313253,0.388723125784971,-0.382371778977509],[0,0,0,0],[8.999999E+09,8.999999E+09,8.999999E+09,8.999999E+09,8.999999E+09,8.999999E+09]];
    LOCAL CONST Robtarget Tr_meulage_motif_1_215 := [[-186.888046875,-18.555173828125,23.7084453125],[0.587839766788017,-0.597604018313253,0.388723125784971,-0.382371778977509],[0,0,0,0],[8.999999E+09,8.999999E+09,8.999999E+09,8.999999E+09,8.999999E+09,8.999999E+09]];
    LOCAL CONST Robtarget Tr_meulage_motif_1_216 := [[-187.259234375,-17.6266171875,23.708443359375],[0.587839766788017,-0.597604018313253,0.388723125784971,-0.382371778977509],[0,0,0,0],[8.999999E+09,8.999999E+09,8.999999E+09,8.999999E+09,8.999999E+09,8.999999E+09]];
    LOCAL CONST Robtarget Tr_meulage_motif_1_217 := [[-187.630421875,-16.69805859375,23.708443359375],[0.587839766788017,-0.597604018313253,0.388723125784971,-0.382371778977509],[0,0,0,0],[8.999999E+09,8.999999E+09,8.999999E+09,8.999999E+09,8.999999E+09,8.999999E+09]];
    LOCAL CONST Robtarget Tr_meulage_motif_1_218 := [[-188.001609375,-15.7695009765625,23.70844140625],[0.587839766788017,-0.597604018313253,0.388723125784971,-0.382371778977509],[0,0,0,0],[8.999999E+09,8.999999E+09,8.999999E+09,8.999999E+09,8.999999E+09,8.999999E+09]];
    LOCAL CONST Robtarget Tr_meulage_motif_1_219 := [[-188.372796875,-14.840943359375,23.70844140625],[0.587839766788017,-0.597604018313253,0.388723125784971,-0.382371778977509],[0,0,0,0],[8.999999E+09,8.999999E+09,8.999999E+09,8.999999E+09,8.999999E+09,8.999999E+09]];
    LOCAL CONST Robtarget Tr_meulage_motif_1_220 := [[-188.743984375,-13.9123857421875,23.70844140625],[0.587839766788017,-0.597604018313253,0.388723125784971,-0.382371778977509],[0,0,0,0],[8.999999E+09,8.999999E+09,8.999999E+09,8.999999E+09,8.999999E+09,8.999999E+09]];
    LOCAL CONST Robtarget Tr_meulage_motif_1_221 := [[-189.115171875,-12.9838271484375,23.708439453125],[0.587839766788017,-0.597604018313253,0.388723125784971,-0.382371778977509],[0,0,0,0],[8.999999E+09,8.999999E+09,8.999999E+09,8.999999E+09,8.999999E+09,8.999999E+09]];
    LOCAL CONST Robtarget Tr_meulage_motif_1_222 := [[-189.486359375,-12.05526953125,23.708439453125],[0.587839766788017,-0.597604018313253,0.388723125784971,-0.382371778977509],[0,0,0,0],[8.999999E+09,8.999999E+09,8.999999E+09,8.999999E+09,8.999999E+09,8.999999E+09]];
    LOCAL CONST Robtarget Tr_meulage_motif_1_223 := [[-189.857546875,-11.1267119140625,23.7084375],[0.587839766788017,-0.597604018313253,0.388723125784971,-0.382371778977509],[0,0,0,0],[8.999999E+09,8.999999E+09,8.999999E+09,8.999999E+09,8.999999E+09,8.999999E+09]];
    LOCAL CONST Robtarget Tr_meulage_motif_1_224 := [[-190.228734375,-10.198154296875,23.7084375],[0.587839766788017,-0.597604018313253,0.388723125784971,-0.382371778977509],[0,0,0,0],[8.999999E+09,8.999999E+09,8.999999E+09,8.999999E+09,8.999999E+09,8.999999E+09]];
    LOCAL CONST Robtarget Tr_meulage_motif_1_225 := [[-190.599921875,-9.2695966796875,23.708435546875],[0.587839766788017,-0.597604018313253,0.388723125784971,-0.382371778977509],[0,0,0,0],[8.999999E+09,8.999999E+09,8.999999E+09,8.999999E+09,8.999999E+09,8.999999E+09]];
    LOCAL CONST Robtarget Tr_meulage_motif_1_226 := [[-190.971109375,-8.3410380859375,23.708435546875],[0.587839766788017,-0.597604018313253,0.388723125784971,-0.382371778977509],[0,0,0,0],[8.999999E+09,8.999999E+09,8.999999E+09,8.999999E+09,8.999999E+09,8.999999E+09]];
    LOCAL CONST Robtarget Tr_meulage_motif_1_227 := [[-191.342296875,-7.41248046875,23.708435546875],[0.587839766788017,-0.597604018313253,0.388723125784971,-0.382371778977509],[0,0,0,0],[8.999999E+09,8.999999E+09,8.999999E+09,8.999999E+09,8.999999E+09,8.999999E+09]];
    LOCAL CONST Robtarget Tr_meulage_motif_1_228 := [[-191.713484375,-6.4839228515625,23.70843359375],[0.587839766788017,-0.597604018313253,0.388723125784971,-0.382371778977509],[0,0,0,0],[8.999999E+09,8.999999E+09,8.999999E+09,8.999999E+09,8.999999E+09,8.999999E+09]];
    LOCAL CONST Robtarget Tr_meulage_motif_1_229 := [[-192.084671875,-5.55536474609375,23.70843359375],[0.587839766788017,-0.597604018313253,0.388723125784971,-0.382371778977509],[0,0,0,0],[8.999999E+09,8.999999E+09,8.999999E+09,8.999999E+09,8.999999E+09,8.999999E+09]];
    LOCAL CONST Robtarget Tr_meulage_motif_1_230 := [[-192.455859375,-4.62680712890625,23.708431640625],[0.587839766788017,-0.597604018313253,0.388723125784971,-0.382371778977509],[0,0,0,0],[8.999999E+09,8.999999E+09,8.999999E+09,8.999999E+09,8.999999E+09,8.999999E+09]];
    LOCAL CONST Robtarget Tr_meulage_motif_1_231 := [[-192.827046875,-3.69824926757813,23.708431640625],[0.587839766788017,-0.597604018313253,0.388723125784971,-0.382371778977509],[0,0,0,0],[8.999999E+09,8.999999E+09,8.999999E+09,8.999999E+09,8.999999E+09,8.999999E+09]];
    LOCAL CONST Robtarget Tr_meulage_motif_1_232 := [[-193.198234375,-2.76969140625,23.708431640625],[0.587839766788017,-0.597604018313253,0.388723125784971,-0.382371778977509],[0,0,0,0],[8.999999E+09,8.999999E+09,8.999999E+09,8.999999E+09,8.999999E+09,8.999999E+09]];
    LOCAL CONST Robtarget Tr_meulage_motif_1_233 := [[-193.569421875,-1.84113366699219,23.7084296875],[0.587839766788017,-0.597604018313253,0.388723125784971,-0.382371778977509],[0,0,0,0],[8.999999E+09,8.999999E+09,8.999999E+09,8.999999E+09,8.999999E+09,8.999999E+09]];
    LOCAL CONST Robtarget Tr_meulage_motif_1_234 := [[-193.940609375,-0.912575866699219,23.7084296875],[0.587839766788017,-0.597604018313253,0.388723125784971,-0.382371778977509],[0,0,0,0],[8.999999E+09,8.999999E+09,8.999999E+09,8.999999E+09,8.999999E+09,8.999999E+09]];
    LOCAL CONST Robtarget Tr_meulage_motif_1_235 := [[-194.311796875,0.015981954574585,23.708427734375],[0.587839766788017,-0.597604018313253,0.388723125784971,-0.382371778977509],[0,0,0,0],[8.999999E+09,8.999999E+09,8.999999E+09,8.999999E+09,8.999999E+09,8.999999E+09]];
    LOCAL CONST Robtarget Tr_meulage_motif_1_236 := [[-194.682984375,0.944539794921875,23.708427734375],[0.587839766788017,-0.597604018313253,0.388723125784971,-0.382371778977509],[0,0,0,0],[8.999999E+09,8.999999E+09,8.999999E+09,8.999999E+09,8.999999E+09,8.999999E+09]];
    LOCAL CONST Robtarget Tr_meulage_motif_1_237 := [[-195.054171875,1.87309765625,23.70842578125],[0.587839766788017,-0.597604018313253,0.388723125784971,-0.382371778977509],[0,0,0,0],[8.999999E+09,8.999999E+09,8.999999E+09,8.999999E+09,8.999999E+09,8.999999E+09]];
    LOCAL CONST Robtarget Tr_meulage_motif_1_238 := [[-195.425359375,2.80165551757813,23.70842578125],[0.587839766788017,-0.597604018313253,0.388723125784971,-0.382371778977509],[0,0,0,0],[8.999999E+09,8.999999E+09,8.999999E+09,8.999999E+09,8.999999E+09,8.999999E+09]];
    LOCAL CONST Robtarget Tr_meulage_motif_1_239 := [[-195.796546875,3.73021313476562,23.70842578125],[0.587839766788017,-0.597604018313253,0.388723125784971,-0.382371778977509],[0,0,0,0],[8.999999E+09,8.999999E+09,8.999999E+09,8.999999E+09,8.999999E+09,8.999999E+09]];
    LOCAL CONST Robtarget Tr_meulage_motif_1_240 := [[-196.167734375,4.65877099609375,23.708423828125],[0.587839766788017,-0.597604018313253,0.388723125784971,-0.382371778977509],[0,0,0,0],[8.999999E+09,8.999999E+09,8.999999E+09,8.999999E+09,8.999999E+09,8.999999E+09]];
    LOCAL CONST Robtarget Tr_meulage_motif_1_241 := [[-196.538921875,5.5873291015625,23.708423828125],[0.587839766788017,-0.597604018313253,0.388723125784971,-0.382371778977509],[0,0,0,0],[8.999999E+09,8.999999E+09,8.999999E+09,8.999999E+09,8.999999E+09,8.999999E+09]];
    LOCAL CONST Robtarget Tr_meulage_motif_1_242 := [[-196.910109375,6.51588671875,23.708421875],[0.587839766788017,-0.597604018313253,0.388723125784971,-0.382371778977509],[0,0,0,0],[8.999999E+09,8.999999E+09,8.999999E+09,8.999999E+09,8.999999E+09,8.999999E+09]];
    LOCAL CONST Robtarget Tr_meulage_motif_1_243 := [[-197.281296875,7.4444443359375,23.708421875],[0.587839766788017,-0.597604018313253,0.388723125784971,-0.382371778977509],[0,0,0,0],[8.999999E+09,8.999999E+09,8.999999E+09,8.999999E+09,8.999999E+09,8.999999E+09]];
    LOCAL CONST Robtarget Tr_meulage_motif_1_244 := [[-197.650859375,8.365642578125,23.597833984375],[0.587839766788017,-0.597604018313253,0.388723125784971,-0.382371778977509],[0,0,0,0],[8.999999E+09,8.999999E+09,8.999999E+09,8.999999E+09,8.999999E+09,8.999999E+09]];
    LOCAL CONST Robtarget Tr_meulage_motif_1_245 := [[-198.004359375,9.2436572265625,23.386658203125],[0.587839766788017,-0.597604018313253,0.388723125784971,-0.382371778977509],[0,0,0,0],[8.999999E+09,8.999999E+09,8.999999E+09,8.999999E+09,8.999999E+09,8.999999E+09]];
    LOCAL CONST Robtarget Tr_meulage_motif_1_246 := [[-198.32365625,10.0343408203125,23.114830078125],[0.587839766788017,-0.597604018313253,0.388723125784971,-0.382371778977509],[0,0,0,0],[8.999999E+09,8.999999E+09,8.999999E+09,8.999999E+09,8.999999E+09,8.999999E+09]];
    LOCAL CONST Robtarget Tr_meulage_motif_1_247 := [[-198.590875,10.6937626953125,22.81070703125],[0.587839766788017,-0.597604018313253,0.388723125784971,-0.382371778977509],[0,0,0,0],[8.999999E+09,8.999999E+09,8.999999E+09,8.999999E+09,8.999999E+09,8.999999E+09]];
    LOCAL CONST Robtarget Tr_meulage_motif_1_248 := [[-198.98165625,11.651611328125,22.148216796875],[0.587839766788017,-0.597604018313253,0.388723125784971,-0.382371778977509],[0,0,0,0],[8.999999E+09,8.999999E+09,8.999999E+09,8.999999E+09,8.999999E+09,8.999999E+09]];
    LOCAL CONST Robtarget Tr_meulage_motif_1_249 := [[-199.3256875,12.4854140625,21.24631640625],[0.587839766788017,-0.597604018313253,0.388723125784971,-0.382371778977509],[0,0,0,0],[8.999999E+09,8.999999E+09,8.999999E+09,8.999999E+09,8.999999E+09,8.999999E+09]];
    LOCAL CONST Robtarget Tr_meulage_motif_1_250 := [[-199.534984375,12.977875,20.200365234375],[0.587839766788017,-0.597604018313253,0.388723125784971,-0.382371778977509],[0,0,0,0],[8.999999E+09,8.999999E+09,8.999999E+09,8.999999E+09,8.999999E+09,8.999999E+09]];
    LOCAL CONST Robtarget Tr_meulage_motif_1_251 := [[-199.6106875,13.14661328125,19.507171875],[0.587839766788017,-0.597604018313253,0.388723125784971,-0.382371778977509],[0,0,0,0],[8.999999E+09,8.999999E+09,8.999999E+09,8.999999E+09,8.999999E+09,8.999999E+09]];
    LOCAL CONST Robtarget Tr_meulage_motif_1_252 := [[-199.64228125,13.2027392578125,18.73721875],[0.587839766788017,-0.597604018313253,0.388723125784971,-0.382371778977509],[0,0,0,0],[8.999999E+09,8.999999E+09,8.999999E+09,8.999999E+09,8.999999E+09,8.999999E+09]];
    LOCAL CONST Robtarget Tr_meulage_motif_1_253 := [[-199.625328125,13.137427734375,17.967408203125],[0.587839766788017,-0.597604018313253,0.388723125784971,-0.382371778977509],[0,0,0,0],[8.999999E+09,8.999999E+09,8.999999E+09,8.999999E+09,8.999999E+09,8.999999E+09]];
    LOCAL CONST Robtarget Tr_meulage_motif_1_254 := [[-199.4809375,12.743267578125,16.859224609375],[0.587839766788017,-0.597604018313253,0.388723125784971,-0.382371778977509],[0,0,0,0],[8.999999E+09,8.999999E+09,8.999999E+09,8.999999E+09,8.999999E+09,8.999999E+09]];
    LOCAL CONST Robtarget Tr_meulage_motif_1_255 := [[-199.33315625,12.3561533203125,16.2735732421875],[0.587839766788017,-0.597604018313253,0.388723125784971,-0.382371778977509],[0,0,0,0],[8.999999E+09,8.999999E+09,8.999999E+09,8.999999E+09,8.999999E+09,8.999999E+09]];
    LOCAL CONST Robtarget Tr_meulage_motif_1_256 := [[-199.01296875,11.5287685546875,15.38647265625],[0.587839766788017,-0.597604018313253,0.388723125784971,-0.382371778977509],[0,0,0,0],[8.999999E+09,8.999999E+09,8.999999E+09,8.999999E+09,8.999999E+09,8.999999E+09]];
    LOCAL CONST Robtarget Tr_meulage_motif_1_257 := [[-198.7998125,10.9832255859375,14.972216796875],[0.587839766788017,-0.597604018313253,0.388723125784971,-0.382371778977509],[0,0,0,0],[8.999999E+09,8.999999E+09,8.999999E+09,8.999999E+09,8.999999E+09,8.999999E+09]];
    LOCAL CONST Robtarget Tr_meulage_motif_1_258 := [[-198.3904375,9.9429541015625,14.4281259765625],[0.587839766788017,-0.597604018313253,0.388723125784971,-0.382371778977509],[0,0,0,0],[8.999999E+09,8.999999E+09,8.999999E+09,8.999999E+09,8.999999E+09,8.999999E+09]];
    LOCAL CONST Robtarget Tr_meulage_motif_1_259 := [[-198.087015625,9.1751318359375,14.13264453125],[0.587839766788017,-0.597604018313253,0.388723125784971,-0.382371778977509],[0,0,0,0],[8.999999E+09,8.999999E+09,8.999999E+09,8.999999E+09,8.999999E+09,8.999999E+09]];
    LOCAL CONST Robtarget Tr_meulage_motif_1_260 := [[-197.743171875,8.308876953125,13.928173828125],[0.587839766788017,-0.597604018313253,0.388723125784971,-0.382371778977509],[0,0,0,0],[8.999999E+09,8.999999E+09,8.999999E+09,8.999999E+09,8.999999E+09,8.999999E+09]];
    LOCAL CONST Robtarget Tr_meulage_motif_1_261 := [[-197.3799375,7.39699462890625,13.8196337890625],[0.587839766788017,-0.597604018313253,0.388723125784971,-0.382371778977509],[0,0,0,0],[8.999999E+09,8.999999E+09,8.999999E+09,8.999999E+09,8.999999E+09,8.999999E+09]];
    LOCAL CONST Robtarget Tr_meulage_motif_1_262 := [[-197.012640625,6.4748896484375,13.7090322265625],[0.587839766788017,-0.597604018313253,0.388723125784971,-0.382371778977509],[0,0,0,0],[8.999999E+09,8.999999E+09,8.999999E+09,8.999999E+09,8.999999E+09,8.999999E+09]];
    LOCAL CONST Robtarget Tr_meulage_motif_1_263 := [[-196.641453125,5.54633154296875,13.709033203125],[0.587839766788017,-0.597604018313253,0.388723125784971,-0.382371778977509],[0,0,0,0],[8.999999E+09,8.999999E+09,8.999999E+09,8.999999E+09,8.999999E+09,8.999999E+09]];
    LOCAL CONST Robtarget Tr_meulage_motif_1_264 := [[-196.270265625,4.61777392578125,13.7090341796875],[0.587839766788017,-0.597604018313253,0.388723125784971,-0.382371778977509],[0,0,0,0],[8.999999E+09,8.999999E+09,8.999999E+09,8.999999E+09,8.999999E+09,8.999999E+09]];
    LOCAL CONST Robtarget Tr_meulage_motif_1_265 := [[-195.899078125,3.68921606445313,13.7090341796875],[0.587839766788017,-0.597604018313253,0.388723125784971,-0.382371778977509],[0,0,0,0],[8.999999E+09,8.999999E+09,8.999999E+09,8.999999E+09,8.999999E+09,8.999999E+09]];
    LOCAL CONST Robtarget Tr_meulage_motif_1_266 := [[-195.527890625,2.760658203125,13.70903515625],[0.587839766788017,-0.597604018313253,0.388723125784971,-0.382371778977509],[0,0,0,0],[8.999999E+09,8.999999E+09,8.999999E+09,8.999999E+09,8.999999E+09,8.999999E+09]];
    LOCAL CONST Robtarget Tr_meulage_motif_1_267 := [[-195.156703125,1.83210046386719,13.7090361328125],[0.587839766788017,-0.597604018313253,0.388723125784971,-0.382371778977509],[0,0,0,0],[8.999999E+09,8.999999E+09,8.999999E+09,8.999999E+09,8.999999E+09,8.999999E+09]];
    LOCAL CONST Robtarget Tr_meulage_motif_1_268 := [[-194.785515625,0.903542602539062,13.709037109375],[0.587839766788017,-0.597604018313253,0.388723125784971,-0.382371778977509],[0,0,0,0],[8.999999E+09,8.999999E+09,8.999999E+09,8.999999E+09,8.999999E+09,8.999999E+09]];
    LOCAL CONST Robtarget Tr_meulage_motif_1_269 := [[-194.414328125,-0.0250152130126953,13.7090380859375],[0.587839766788017,-0.597604018313253,0.388723125784971,-0.382371778977509],[0,0,0,0],[8.999999E+09,8.999999E+09,8.999999E+09,8.999999E+09,8.999999E+09,8.999999E+09]];
    LOCAL CONST Robtarget Tr_meulage_motif_1_270 := [[-194.043140625,-0.953573059082031,13.7090390625],[0.587839766788017,-0.597604018313253,0.388723125784971,-0.382371778977509],[0,0,0,0],[8.999999E+09,8.999999E+09,8.999999E+09,8.999999E+09,8.999999E+09,8.999999E+09]];
    LOCAL CONST Robtarget Tr_meulage_motif_1_271 := [[-193.671953125,-1.882130859375,13.7090400390625],[0.587839766788017,-0.597604018313253,0.388723125784971,-0.382371778977509],[0,0,0,0],[8.999999E+09,8.999999E+09,8.999999E+09,8.999999E+09,8.999999E+09,8.999999E+09]];
    LOCAL CONST Robtarget Tr_meulage_motif_1_272 := [[-193.300765625,-2.81068872070313,13.7090400390625],[0.587839766788017,-0.597604018313253,0.388723125784971,-0.382371778977509],[0,0,0,0],[8.999999E+09,8.999999E+09,8.999999E+09,8.999999E+09,8.999999E+09,8.999999E+09]];
    LOCAL CONST Robtarget Tr_meulage_motif_1_273 := [[-192.929578125,-3.73924658203125,13.709041015625],[0.587839766788017,-0.597604018313253,0.388723125784971,-0.382371778977509],[0,0,0,0],[8.999999E+09,8.999999E+09,8.999999E+09,8.999999E+09,8.999999E+09,8.999999E+09]];
    LOCAL CONST Robtarget Tr_meulage_motif_1_274 := [[-192.558390625,-4.66780419921875,13.7090419921875],[0.587839766788017,-0.597604018313253,0.388723125784971,-0.382371778977509],[0,0,0,0],[8.999999E+09,8.999999E+09,8.999999E+09,8.999999E+09,8.999999E+09,8.999999E+09]];
    LOCAL CONST Robtarget Tr_meulage_motif_1_275 := [[-192.187203125,-5.5963623046875,13.70904296875],[0.587839766788017,-0.597604018313253,0.388723125784971,-0.382371778977509],[0,0,0,0],[8.999999E+09,8.999999E+09,8.999999E+09,8.999999E+09,8.999999E+09,8.999999E+09]];
    LOCAL CONST Robtarget Tr_meulage_motif_1_276 := [[-191.816015625,-6.524919921875,13.7090439453125],[0.587839766788017,-0.597604018313253,0.388723125784971,-0.382371778977509],[0,0,0,0],[8.999999E+09,8.999999E+09,8.999999E+09,8.999999E+09,8.999999E+09,8.999999E+09]];
    LOCAL CONST Robtarget Tr_meulage_motif_1_277 := [[-191.444828125,-7.45347802734375,13.709044921875],[0.587839766788017,-0.597604018313253,0.388723125784971,-0.382371778977509],[0,0,0,0],[8.999999E+09,8.999999E+09,8.999999E+09,8.999999E+09,8.999999E+09,8.999999E+09]];
    LOCAL CONST Robtarget Tr_meulage_motif_1_278 := [[-191.073640625,-8.38203515625,13.709044921875],[0.587839766788017,-0.597604018313253,0.388723125784971,-0.382371778977509],[0,0,0,0],[8.999999E+09,8.999999E+09,8.999999E+09,8.999999E+09,8.999999E+09,8.999999E+09]];
    LOCAL CONST Robtarget Tr_meulage_motif_1_279 := [[-190.702453125,-9.31059375,13.7090458984375],[0.587839766788017,-0.597604018313253,0.388723125784971,-0.382371778977509],[0,0,0,0],[8.999999E+09,8.999999E+09,8.999999E+09,8.999999E+09,8.999999E+09,8.999999E+09]];
    LOCAL CONST Robtarget Tr_meulage_motif_1_280 := [[-190.331265625,-10.2391513671875,13.709046875],[0.587839766788017,-0.597604018313253,0.388723125784971,-0.382371778977509],[0,0,0,0],[8.999999E+09,8.999999E+09,8.999999E+09,8.999999E+09,8.999999E+09,8.999999E+09]];
    LOCAL CONST Robtarget Tr_meulage_motif_1_281 := [[-189.960078125,-11.167708984375,13.7090478515625],[0.587839766788017,-0.597604018313253,0.388723125784971,-0.382371778977509],[0,0,0,0],[8.999999E+09,8.999999E+09,8.999999E+09,8.999999E+09,8.999999E+09,8.999999E+09]];
    LOCAL CONST Robtarget Tr_meulage_motif_1_282 := [[-189.588890625,-12.0962666015625,13.709048828125],[0.587839766788017,-0.597604018313253,0.388723125784971,-0.382371778977509],[0,0,0,0],[8.999999E+09,8.999999E+09,8.999999E+09,8.999999E+09,8.999999E+09,8.999999E+09]];
    LOCAL CONST Robtarget Tr_meulage_motif_1_283 := [[-189.217703125,-13.0248251953125,13.7090498046875],[0.587839766788017,-0.597604018313253,0.388723125784971,-0.382371778977509],[0,0,0,0],[8.999999E+09,8.999999E+09,8.999999E+09,8.999999E+09,8.999999E+09,8.999999E+09]];
    LOCAL CONST Robtarget Tr_meulage_motif_1_284 := [[-188.846515625,-13.9533828125,13.7090498046875],[0.587839766788017,-0.597604018313253,0.388723125784971,-0.382371778977509],[0,0,0,0],[8.999999E+09,8.999999E+09,8.999999E+09,8.999999E+09,8.999999E+09,8.999999E+09]];
    LOCAL CONST Robtarget Tr_meulage_motif_1_285 := [[-188.475328125,-14.8819404296875,13.70905078125],[0.587839766788017,-0.597604018313253,0.388723125784971,-0.382371778977509],[0,0,0,0],[8.999999E+09,8.999999E+09,8.999999E+09,8.999999E+09,8.999999E+09,8.999999E+09]];
    LOCAL CONST Robtarget Tr_meulage_motif_1_286 := [[-188.104140625,-15.810498046875,13.7090517578125],[0.587839766788017,-0.597604018313253,0.388723125784971,-0.382371778977509],[0,0,0,0],[8.999999E+09,8.999999E+09,8.999999E+09,8.999999E+09,8.999999E+09,8.999999E+09]];
    LOCAL CONST Robtarget Tr_meulage_motif_1_287 := [[-187.732953125,-16.739056640625,13.709052734375],[0.587839766788017,-0.597604018313253,0.388723125784971,-0.382371778977509],[0,0,0,0],[8.999999E+09,8.999999E+09,8.999999E+09,8.999999E+09,8.999999E+09,8.999999E+09]];
    LOCAL CONST Robtarget Tr_meulage_motif_1_288 := [[-187.361765625,-17.66761328125,13.7090537109375],[0.587839766788017,-0.597604018313253,0.388723125784971,-0.382371778977509],[0,0,0,0],[8.999999E+09,8.999999E+09,8.999999E+09,8.999999E+09,8.999999E+09,8.999999E+09]];
    LOCAL CONST Robtarget Tr_meulage_motif_1_289 := [[-186.990578125,-18.596171875,13.7090546875],[0.587839766788017,-0.597604018313253,0.388723125784971,-0.382371778977509],[0,0,0,0],[8.999999E+09,8.999999E+09,8.999999E+09,8.999999E+09,8.999999E+09,8.999999E+09]];
    LOCAL CONST Robtarget Tr_meulage_motif_1_290 := [[-186.619390625,-19.524728515625,13.7090556640625],[0.587839766788017,-0.597604018313253,0.388723125784971,-0.382371778977509],[0,0,0,0],[8.999999E+09,8.999999E+09,8.999999E+09,8.999999E+09,8.999999E+09,8.999999E+09]];
    LOCAL CONST Robtarget Tr_meulage_motif_1_291 := [[-186.248203125,-20.453287109375,13.7090556640625],[0.587839766788017,-0.597604018313253,0.388723125784971,-0.382371778977509],[0,0,0,0],[8.999999E+09,8.999999E+09,8.999999E+09,8.999999E+09,8.999999E+09,8.999999E+09]];
    LOCAL CONST Robtarget Tr_meulage_motif_1_292 := [[-185.877015625,-21.381845703125,13.709056640625],[0.587839766788017,-0.597604018313253,0.388723125784971,-0.382371778977509],[0,0,0,0],[8.999999E+09,8.999999E+09,8.999999E+09,8.999999E+09,8.999999E+09,8.999999E+09]];
    LOCAL CONST Robtarget Tr_meulage_motif_1_293 := [[-185.505828125,-22.31040234375,13.7090576171875],[0.587839766788017,-0.597604018313253,0.388723125784971,-0.382371778977509],[0,0,0,0],[8.999999E+09,8.999999E+09,8.999999E+09,8.999999E+09,8.999999E+09,8.999999E+09]];
    LOCAL CONST Robtarget Tr_meulage_motif_1_294 := [[-185.134640625,-23.2389609375,13.70905859375],[0.587839766788017,-0.597604018313253,0.388723125784971,-0.382371778977509],[0,0,0,0],[8.999999E+09,8.999999E+09,8.999999E+09,8.999999E+09,8.999999E+09,8.999999E+09]];
    LOCAL CONST Robtarget Tr_meulage_motif_1_295 := [[-184.763453125,-24.16751953125,13.7090595703125],[0.587839766788017,-0.597604018313253,0.388723125784971,-0.382371778977509],[0,0,0,0],[8.999999E+09,8.999999E+09,8.999999E+09,8.999999E+09,8.999999E+09,8.999999E+09]];
    LOCAL CONST Robtarget Tr_meulage_motif_1_296 := [[-184.392265625,-25.096076171875,13.709060546875],[0.587839766788017,-0.597604018313253,0.388723125784971,-0.382371778977509],[0,0,0,0],[8.999999E+09,8.999999E+09,8.999999E+09,8.999999E+09,8.999999E+09,8.999999E+09]];
    LOCAL CONST Robtarget Tr_meulage_motif_1_297 := [[-184.021078125,-26.024634765625,13.709060546875],[0.587839766788017,-0.597604018313253,0.388723125784971,-0.382371778977509],[0,0,0,0],[8.999999E+09,8.999999E+09,8.999999E+09,8.999999E+09,8.999999E+09,8.999999E+09]];
    LOCAL CONST Robtarget Tr_meulage_motif_1_298 := [[-183.649890625,-26.95319140625,13.7090615234375],[0.587839766788017,-0.597604018313253,0.388723125784971,-0.382371778977509],[0,0,0,0],[8.999999E+09,8.999999E+09,8.999999E+09,8.999999E+09,8.999999E+09,8.999999E+09]];
    LOCAL CONST Robtarget Tr_meulage_motif_1_299 := [[-183.278703125,-27.88175,13.7090625],[0.587839766788017,-0.597604018313253,0.388723125784971,-0.382371778977509],[0,0,0,0],[8.999999E+09,8.999999E+09,8.999999E+09,8.999999E+09,8.999999E+09,8.999999E+09]];
    LOCAL CONST Robtarget Tr_meulage_motif_1_300 := [[-182.907515625,-28.81030859375,13.7090634765625],[0.587839766788017,-0.597604018313253,0.388723125784971,-0.382371778977509],[0,0,0,0],[8.999999E+09,8.999999E+09,8.999999E+09,8.999999E+09,8.999999E+09,8.999999E+09]];
    LOCAL CONST Robtarget Tr_meulage_motif_1_301 := [[-182.536328125,-29.738865234375,13.709064453125],[0.587839766788017,-0.597604018313253,0.388723125784971,-0.382371778977509],[0,0,0,0],[8.999999E+09,8.999999E+09,8.999999E+09,8.999999E+09,8.999999E+09,8.999999E+09]];
    LOCAL CONST Robtarget Tr_meulage_motif_1_302 := [[-182.165140625,-30.667423828125,13.7090654296875],[0.587839766788017,-0.597604018313253,0.388723125784971,-0.382371778977509],[0,0,0,0],[8.999999E+09,8.999999E+09,8.999999E+09,8.999999E+09,8.999999E+09,8.999999E+09]];
    LOCAL CONST Robtarget Tr_meulage_motif_1_303 := [[-181.793953125,-31.59598046875,13.7090654296875],[0.587839766788017,-0.597604018313253,0.388723125784971,-0.382371778977509],[0,0,0,0],[8.999999E+09,8.999999E+09,8.999999E+09,8.999999E+09,8.999999E+09,8.999999E+09]];
    LOCAL CONST Robtarget Tr_meulage_motif_1_304 := [[-181.422765625,-32.5245390625,13.70906640625],[0.587839766788017,-0.597604018313253,0.388723125784971,-0.382371778977509],[0,0,0,0],[8.999999E+09,8.999999E+09,8.999999E+09,8.999999E+09,8.999999E+09,8.999999E+09]];
    LOCAL CONST Robtarget Tr_meulage_motif_1_305 := [[-181.051578125,-33.45309765625,13.7090673828125],[0.587839766788017,-0.597604018313253,0.388723125784971,-0.382371778977509],[0,0,0,0],[8.999999E+09,8.999999E+09,8.999999E+09,8.999999E+09,8.999999E+09,8.999999E+09]];
    LOCAL CONST Robtarget Tr_meulage_motif_1_306 := [[-180.680390625,-34.38165625,13.709068359375],[0.587839766788017,-0.597604018313253,0.388723125784971,-0.382371778977509],[0,0,0,0],[8.999999E+09,8.999999E+09,8.999999E+09,8.999999E+09,8.999999E+09,8.999999E+09]];
    LOCAL CONST Robtarget Tr_meulage_motif_1_307 := [[-180.31309375,-35.3037578125,13.598466796875],[0.587839766788017,-0.597604018313253,0.388723125784971,-0.382371778977509],[0,0,0,0],[8.999999E+09,8.999999E+09,8.999999E+09,8.999999E+09,8.999999E+09,8.999999E+09]];
    LOCAL CONST Robtarget Tr_meulage_motif_1_308 := [[-179.963921875,-36.18350390625,13.38729296875],[0.587839766788017,-0.597604018313253,0.388723125784971,-0.382371778977509],[0,0,0,0],[8.999999E+09,8.999999E+09,8.999999E+09,8.999999E+09,8.999999E+09,8.999999E+09]];
    LOCAL CONST Robtarget Tr_meulage_motif_1_309 := [[-179.650203125,-36.97641796875,13.1154814453125],[0.587839766788017,-0.597604018313253,0.388723125784971,-0.382371778977509],[0,0,0,0],[8.999999E+09,8.999999E+09,8.999999E+09,8.999999E+09,8.999999E+09,8.999999E+09]];
    LOCAL CONST Robtarget Tr_meulage_motif_1_310 := [[-179.37465625,-37.67391015625,12.8395615234375],[0.587839766788017,-0.597604018313253,0.388723125784971,-0.382371778977509],[0,0,0,0],[8.999999E+09,8.999999E+09,8.999999E+09,8.999999E+09,8.999999E+09,8.999999E+09]];
    LOCAL CONST Robtarget Tr_meulage_motif_1_311 := [[-178.97228125,-38.6988359375,12.2234755859375],[0.587839766788017,-0.597604018313253,0.388723125784971,-0.382371778977509],[0,0,0,0],[8.999999E+09,8.999999E+09,8.999999E+09,8.999999E+09,8.999999E+09,8.999999E+09]];
    LOCAL CONST Robtarget Tr_meulage_motif_1_312 := [[-178.600921875,-39.6530390625,11.37588671875],[0.587839766788017,-0.597604018313253,0.388723125784971,-0.382371778977509],[0,0,0,0],[8.999999E+09,8.999999E+09,8.999999E+09,8.999999E+09,8.999999E+09,8.999999E+09]];
    LOCAL CONST Robtarget Tr_meulage_motif_1_313 := [[-178.29678125,-40.44433203125,10.3520908203125],[0.587839766788017,-0.597604018313253,0.388723125784971,-0.382371778977509],[0,0,0,0],[8.999999E+09,8.999999E+09,8.999999E+09,8.999999E+09,8.999999E+09,8.999999E+09]];
    LOCAL CONST Robtarget Tr_meulage_motif_1_314 := [[-178.127015625,-40.90219140625,9.2359248046875],[0.587839766788017,-0.597604018313253,0.388723125784971,-0.382371778977509],[0,0,0,0],[8.999999E+09,8.999999E+09,8.999999E+09,8.999999E+09,8.999999E+09,8.999999E+09]];
    LOCAL CONST Robtarget Tr_meulage_motif_1_315 := [[-178.124109375,-40.930171875,8.5400302734375],[0.587839766788017,-0.597604018313253,0.388723125784971,-0.382371778977509],[0,0,0,0],[8.999999E+09,8.999999E+09,8.999999E+09,8.999999E+09,8.999999E+09,8.999999E+09]];
    LOCAL CONST Robtarget Tr_meulage_motif_1_316 := [[-178.130890625,-40.93288671875,7.8787890625],[0.587839766788017,-0.597604018313253,0.388723125784971,-0.382371778977509],[0,0,0,0],[8.999999E+09,8.999999E+09,8.999999E+09,8.999999E+09,8.999999E+09,8.999999E+09]];
    LOCAL CONST Robtarget Tr_meulage_motif_1_317 := [[-178.158046875,-40.884640625,7.2177509765625],[0.587839766788017,-0.597604018313253,0.388723125784971,-0.382371778977509],[0,0,0,0],[8.999999E+09,8.999999E+09,8.999999E+09,8.999999E+09,8.999999E+09,8.999999E+09]];
    LOCAL CONST Robtarget Tr_meulage_motif_1_318 := [[-178.354265625,-40.42653125,6.11608349609375],[0.587839766788017,-0.597604018313253,0.388723125784971,-0.382371778977509],[0,0,0,0],[8.999999E+09,8.999999E+09,8.999999E+09,8.999999E+09,8.999999E+09,8.999999E+09]];
    LOCAL CONST Robtarget Tr_meulage_motif_1_319 := [[-178.6825625,-39.635234375,5.10950341796875],[0.587839766788017,-0.597604018313253,0.388723125784971,-0.382371778977509],[0,0,0,0],[8.999999E+09,8.999999E+09,8.999999E+09,8.999999E+09,8.999999E+09,8.999999E+09]];
    LOCAL CONST Robtarget Tr_meulage_motif_1_320 := [[-179.0709375,-38.68833984375,4.28069384765625],[0.587839766788017,-0.597604018313253,0.388723125784971,-0.382371778977509],[0,0,0,0],[8.999999E+09,8.999999E+09,8.999999E+09,8.999999E+09,8.999999E+09,8.999999E+09]];
    LOCAL CONST Robtarget Tr_meulage_motif_1_321 := [[-179.33003125,-38.05195703125,3.88495190429688],[0.587839766788017,-0.597604018313253,0.388723125784971,-0.382371778977509],[0,0,0,0],[8.999999E+09,8.999999E+09,8.999999E+09,8.999999E+09,8.999999E+09,8.999999E+09]];
    LOCAL CONST Robtarget Tr_meulage_motif_1_322 := [[-179.764921875,-36.9785390625,3.39744946289062],[0.587839766788017,-0.597604018313253,0.388723125784971,-0.382371778977509],[0,0,0,0],[8.999999E+09,8.999999E+09,8.999999E+09,8.999999E+09,8.999999E+09,8.999999E+09]];
    LOCAL CONST Robtarget Tr_meulage_motif_1_323 := [[-180.081296875,-36.1949609375,3.13335546875],[0.587839766788017,-0.597604018313253,0.388723125784971,-0.382371778977509],[0,0,0,0],[8.999999E+09,8.999999E+09,8.999999E+09,8.999999E+09,8.999999E+09,8.999999E+09]];
    LOCAL CONST Robtarget Tr_meulage_motif_1_324 := [[-180.42934375,-35.3303828125,2.9288828125],[0.587839766788017,-0.597604018313253,0.388723125784971,-0.382371778977509],[0,0,0,0],[8.999999E+09,8.999999E+09,8.999999E+09,8.999999E+09,8.999999E+09,8.999999E+09]];
    LOCAL CONST Robtarget Tr_meulage_motif_1_325 := [[-180.794796875,-34.419390625,2.820341796875],[0.587839766788017,-0.597604018313253,0.388723125784971,-0.382371778977509],[0,0,0,0],[8.999999E+09,8.999999E+09,8.999999E+09,8.999999E+09,8.999999E+09,8.999999E+09]];
    LOCAL CONST Robtarget Tr_meulage_motif_1_326 := [[-181.164359375,-33.4981953125,2.70973828125],[0.587839766788017,-0.597604018313253,0.388723125784971,-0.382371778977509],[0,0,0,0],[8.999999E+09,8.999999E+09,8.999999E+09,8.999999E+09,8.999999E+09,8.999999E+09]];
    LOCAL CONST Robtarget Tr_meulage_motif_1_327 := [[-181.535546875,-32.56963671875,2.70973754882813],[0.587839766788017,-0.597604018313253,0.388723125784971,-0.382371778977509],[0,0,0,0],[8.999999E+09,8.999999E+09,8.999999E+09,8.999999E+09,8.999999E+09,8.999999E+09]];
    LOCAL CONST Robtarget Tr_meulage_motif_1_328 := [[-181.906734375,-31.641078125,2.70973657226563],[0.587839766788017,-0.597604018313253,0.388723125784971,-0.382371778977509],[0,0,0,0],[8.999999E+09,8.999999E+09,8.999999E+09,8.999999E+09,8.999999E+09,8.999999E+09]];
    LOCAL CONST Robtarget Tr_meulage_motif_1_329 := [[-182.277921875,-30.71251953125,2.70973583984375],[0.587839766788017,-0.597604018313253,0.388723125784971,-0.382371778977509],[0,0,0,0],[8.999999E+09,8.999999E+09,8.999999E+09,8.999999E+09,8.999999E+09,8.999999E+09]];
    LOCAL CONST Robtarget Tr_meulage_motif_1_330 := [[-182.649109375,-29.783962890625,2.70973486328125],[0.587839766788017,-0.597604018313253,0.388723125784971,-0.382371778977509],[0,0,0,0],[8.999999E+09,8.999999E+09,8.999999E+09,8.999999E+09,8.999999E+09,8.999999E+09]];
    LOCAL CONST Robtarget Tr_meulage_motif_1_331 := [[-183.020296875,-28.855404296875,2.70973413085937],[0.587839766788017,-0.597604018313253,0.388723125784971,-0.382371778977509],[0,0,0,0],[8.999999E+09,8.999999E+09,8.999999E+09,8.999999E+09,8.999999E+09,8.999999E+09]];
    LOCAL CONST Robtarget Tr_meulage_motif_1_332 := [[-183.391484375,-27.92684765625,2.7097333984375],[0.587839766788017,-0.597604018313253,0.388723125784971,-0.382371778977509],[0,0,0,0],[8.999999E+09,8.999999E+09,8.999999E+09,8.999999E+09,8.999999E+09,8.999999E+09]];
    LOCAL CONST Robtarget Tr_meulage_motif_1_333 := [[-183.762671875,-26.9982890625,2.709732421875],[0.587839766788017,-0.597604018313253,0.388723125784971,-0.382371778977509],[0,0,0,0],[8.999999E+09,8.999999E+09,8.999999E+09,8.999999E+09,8.999999E+09,8.999999E+09]];
    LOCAL CONST Robtarget Tr_meulage_motif_1_334 := [[-184.133859375,-26.06973046875,2.70973168945312],[0.587839766788017,-0.597604018313253,0.388723125784971,-0.382371778977509],[0,0,0,0],[8.999999E+09,8.999999E+09,8.999999E+09,8.999999E+09,8.999999E+09,8.999999E+09]];
    LOCAL CONST Robtarget Tr_meulage_motif_1_335 := [[-184.505046875,-25.141173828125,2.70973095703125],[0.587839766788017,-0.597604018313253,0.388723125784971,-0.382371778977509],[0,0,0,0],[8.999999E+09,8.999999E+09,8.999999E+09,8.999999E+09,8.999999E+09,8.999999E+09]];
    LOCAL CONST Robtarget Tr_meulage_motif_1_336 := [[-184.876234375,-24.212615234375,2.70972998046875],[0.587839766788017,-0.597604018313253,0.388723125784971,-0.382371778977509],[0,0,0,0],[8.999999E+09,8.999999E+09,8.999999E+09,8.999999E+09,8.999999E+09,8.999999E+09]];
    LOCAL CONST Robtarget Tr_meulage_motif_1_337 := [[-185.247421875,-23.28405859375,2.70972924804687],[0.587839766788017,-0.597604018313253,0.388723125784971,-0.382371778977509],[0,0,0,0],[8.999999E+09,8.999999E+09,8.999999E+09,8.999999E+09,8.999999E+09,8.999999E+09]];
    LOCAL CONST Robtarget Tr_meulage_motif_1_338 := [[-185.618609375,-22.3555,2.70972827148438],[0.587839766788017,-0.597604018313253,0.388723125784971,-0.382371778977509],[0,0,0,0],[8.999999E+09,8.999999E+09,8.999999E+09,8.999999E+09,8.999999E+09,8.999999E+09]];
    LOCAL CONST Robtarget Tr_meulage_motif_1_339 := [[-185.989796875,-21.42694140625,2.7097275390625],[0.587839766788017,-0.597604018313253,0.388723125784971,-0.382371778977509],[0,0,0,0],[8.999999E+09,8.999999E+09,8.999999E+09,8.999999E+09,8.999999E+09,8.999999E+09]];
    LOCAL CONST Robtarget Tr_meulage_motif_1_340 := [[-186.360984375,-20.498384765625,2.70972680664063],[0.587839766788017,-0.597604018313253,0.388723125784971,-0.382371778977509],[0,0,0,0],[8.999999E+09,8.999999E+09,8.999999E+09,8.999999E+09,8.999999E+09,8.999999E+09]];
    LOCAL CONST Robtarget Tr_meulage_motif_1_341 := [[-186.732171875,-19.569826171875,2.70972583007813],[0.587839766788017,-0.597604018313253,0.388723125784971,-0.382371778977509],[0,0,0,0],[8.999999E+09,8.999999E+09,8.999999E+09,8.999999E+09,8.999999E+09,8.999999E+09]];
    LOCAL CONST Robtarget Tr_meulage_motif_1_342 := [[-187.103359375,-18.641267578125,2.70972509765625],[0.587839766788017,-0.597604018313253,0.388723125784971,-0.382371778977509],[0,0,0,0],[8.999999E+09,8.999999E+09,8.999999E+09,8.999999E+09,8.999999E+09,8.999999E+09]];
    LOCAL CONST Robtarget Tr_meulage_motif_1_343 := [[-187.474546875,-17.7127109375,2.70972436523438],[0.587839766788017,-0.597604018313253,0.388723125784971,-0.382371778977509],[0,0,0,0],[8.999999E+09,8.999999E+09,8.999999E+09,8.999999E+09,8.999999E+09,8.999999E+09]];
    LOCAL CONST Robtarget Tr_meulage_motif_1_344 := [[-187.845734375,-16.78415234375,2.70972338867188],[0.587839766788017,-0.597604018313253,0.388723125784971,-0.382371778977509],[0,0,0,0],[8.999999E+09,8.999999E+09,8.999999E+09,8.999999E+09,8.999999E+09,8.999999E+09]];
    LOCAL CONST Robtarget Tr_meulage_motif_1_345 := [[-188.2169375,-15.8555947265625,2.70972265625],[0.587839766788017,-0.597604018313253,0.388723125784971,-0.382371778977509],[0,0,0,0],[8.999999E+09,8.999999E+09,8.999999E+09,8.999999E+09,8.999999E+09,8.999999E+09]];
    LOCAL CONST Robtarget Tr_meulage_motif_1_346 := [[-188.588125,-14.927037109375,2.70972192382813],[0.587839766788017,-0.597604018313253,0.388723125784971,-0.382371778977509],[0,0,0,0],[8.999999E+09,8.999999E+09,8.999999E+09,8.999999E+09,8.999999E+09,8.999999E+09]];
    LOCAL CONST Robtarget Tr_meulage_motif_1_347 := [[-188.9593125,-13.9984794921875,2.70972094726562],[0.587839766788017,-0.597604018313253,0.388723125784971,-0.382371778977509],[0,0,0,0],[8.999999E+09,8.999999E+09,8.999999E+09,8.999999E+09,8.999999E+09,8.999999E+09]];
    LOCAL CONST Robtarget Tr_meulage_motif_1_348 := [[-189.3305,-13.069921875,2.70972021484375],[0.587839766788017,-0.597604018313253,0.388723125784971,-0.382371778977509],[0,0,0,0],[8.999999E+09,8.999999E+09,8.999999E+09,8.999999E+09,8.999999E+09,8.999999E+09]];
    LOCAL CONST Robtarget Tr_meulage_motif_1_349 := [[-189.7016875,-12.1413642578125,2.70971923828125],[0.587839766788017,-0.597604018313253,0.388723125784971,-0.382371778977509],[0,0,0,0],[8.999999E+09,8.999999E+09,8.999999E+09,8.999999E+09,8.999999E+09,8.999999E+09]];
    LOCAL CONST Robtarget Tr_meulage_motif_1_350 := [[-190.072875,-11.2128056640625,2.70971850585937],[0.587839766788017,-0.597604018313253,0.388723125784971,-0.382371778977509],[0,0,0,0],[8.999999E+09,8.999999E+09,8.999999E+09,8.999999E+09,8.999999E+09,8.999999E+09]];
    LOCAL CONST Robtarget Tr_meulage_motif_1_351 := [[-190.4440625,-10.284248046875,2.7097177734375],[0.587839766788017,-0.597604018313253,0.388723125784971,-0.382371778977509],[0,0,0,0],[8.999999E+09,8.999999E+09,8.999999E+09,8.999999E+09,8.999999E+09,8.999999E+09]];
    LOCAL CONST Robtarget Tr_meulage_motif_1_352 := [[-190.81525,-9.3556904296875,2.709716796875],[0.587839766788017,-0.597604018313253,0.388723125784971,-0.382371778977509],[0,0,0,0],[8.999999E+09,8.999999E+09,8.999999E+09,8.999999E+09,8.999999E+09,8.999999E+09]];
    LOCAL CONST Robtarget Tr_meulage_motif_1_353 := [[-191.1864375,-8.4271328125,2.70971606445312],[0.587839766788017,-0.597604018313253,0.388723125784971,-0.382371778977509],[0,0,0,0],[8.999999E+09,8.999999E+09,8.999999E+09,8.999999E+09,8.999999E+09,8.999999E+09]];
    LOCAL CONST Robtarget Tr_meulage_motif_1_354 := [[-191.557625,-7.49857470703125,2.70971533203125],[0.587839766788017,-0.597604018313253,0.388723125784971,-0.382371778977509],[0,0,0,0],[8.999999E+09,8.999999E+09,8.999999E+09,8.999999E+09,8.999999E+09,8.999999E+09]];
    LOCAL CONST Robtarget Tr_meulage_motif_1_355 := [[-191.9288125,-6.57001708984375,2.70971435546875],[0.587839766788017,-0.597604018313253,0.388723125784971,-0.382371778977509],[0,0,0,0],[8.999999E+09,8.999999E+09,8.999999E+09,8.999999E+09,8.999999E+09,8.999999E+09]];
    LOCAL CONST Robtarget Tr_meulage_motif_1_356 := [[-192.3,-5.641458984375,2.70971362304688],[0.587839766788017,-0.597604018313253,0.388723125784971,-0.382371778977509],[0,0,0,0],[8.999999E+09,8.999999E+09,8.999999E+09,8.999999E+09,8.999999E+09,8.999999E+09]];
    LOCAL CONST Robtarget Tr_meulage_motif_1_357 := [[-192.6711875,-4.7129013671875,2.70971264648438],[0.587839766788017,-0.597604018313253,0.388723125784971,-0.382371778977509],[0,0,0,0],[8.999999E+09,8.999999E+09,8.999999E+09,8.999999E+09,8.999999E+09,8.999999E+09]];
    LOCAL CONST Robtarget Tr_meulage_motif_1_358 := [[-193.042375,-3.78434350585938,2.7097119140625],[0.587839766788017,-0.597604018313253,0.388723125784971,-0.382371778977509],[0,0,0,0],[8.999999E+09,8.999999E+09,8.999999E+09,8.999999E+09,8.999999E+09,8.999999E+09]];
    LOCAL CONST Robtarget Tr_meulage_motif_1_359 := [[-193.4135625,-2.85578564453125,2.70971118164063],[0.587839766788017,-0.597604018313253,0.388723125784971,-0.382371778977509],[0,0,0,0],[8.999999E+09,8.999999E+09,8.999999E+09,8.999999E+09,8.999999E+09,8.999999E+09]];
    LOCAL CONST Robtarget Tr_meulage_motif_1_360 := [[-193.78475,-1.92722778320313,2.70971020507812],[0.587839766788017,-0.597604018313253,0.388723125784971,-0.382371778977509],[0,0,0,0],[8.999999E+09,8.999999E+09,8.999999E+09,8.999999E+09,8.999999E+09,8.999999E+09]];
    LOCAL CONST Robtarget Tr_meulage_motif_1_361 := [[-194.1559375,-0.998669921875,2.70970947265625],[0.587839766788017,-0.597604018313253,0.388723125784971,-0.382371778977509],[0,0,0,0],[8.999999E+09,8.999999E+09,8.999999E+09,8.999999E+09,8.999999E+09,8.999999E+09]];
    LOCAL CONST Robtarget Tr_meulage_motif_1_362 := [[-194.527125,-0.0701120986938477,2.70970874023438],[0.587839766788017,-0.597604018313253,0.388723125784971,-0.382371778977509],[0,0,0,0],[8.999999E+09,8.999999E+09,8.999999E+09,8.999999E+09,8.999999E+09,8.999999E+09]];
    LOCAL CONST Robtarget Tr_meulage_motif_1_363 := [[-194.8983125,0.858445739746094,2.70970776367187],[0.587839766788017,-0.597604018313253,0.388723125784971,-0.382371778977509],[0,0,0,0],[8.999999E+09,8.999999E+09,8.999999E+09,8.999999E+09,8.999999E+09,8.999999E+09]];
    LOCAL CONST Robtarget Tr_meulage_motif_1_364 := [[-195.2695,1.78700354003906,2.70970703125],[0.587839766788017,-0.597604018313253,0.388723125784971,-0.382371778977509],[0,0,0,0],[8.999999E+09,8.999999E+09,8.999999E+09,8.999999E+09,8.999999E+09,8.999999E+09]];
    LOCAL CONST Robtarget Tr_meulage_motif_1_365 := [[-195.6406875,2.71556127929688,2.7097060546875],[0.587839766788017,-0.597604018313253,0.388723125784971,-0.382371778977509],[0,0,0,0],[8.999999E+09,8.999999E+09,8.999999E+09,8.999999E+09,8.999999E+09,8.999999E+09]];
    LOCAL CONST Robtarget Tr_meulage_motif_1_366 := [[-196.011875,3.644119140625,2.70970532226562],[0.587839766788017,-0.597604018313253,0.388723125784971,-0.382371778977509],[0,0,0,0],[8.999999E+09,8.999999E+09,8.999999E+09,8.999999E+09,8.999999E+09,8.999999E+09]];
    LOCAL CONST Robtarget Tr_meulage_motif_1_367 := [[-196.3830625,4.57267724609375,2.70970458984375],[0.587839766788017,-0.597604018313253,0.388723125784971,-0.382371778977509],[0,0,0,0],[8.999999E+09,8.999999E+09,8.999999E+09,8.999999E+09,8.999999E+09,8.999999E+09]];
    LOCAL CONST Robtarget Tr_meulage_motif_1_368 := [[-196.75425,5.50123486328125,2.70970361328125],[0.587839766788017,-0.597604018313253,0.388723125784971,-0.382371778977509],[0,0,0,0],[8.999999E+09,8.999999E+09,8.999999E+09,8.999999E+09,8.999999E+09,8.999999E+09]];
